// TIA Portal project "Proyecto_Automatizacion" (V18)

(* hardware
DEVICE "S7-1500/ET200MP station_1"  S7-1500 station
   slot 0: "Rail_0"  Rack  6ES7 590-1***0-0AA0
   slot 1: "Celda_Mecanizado"  CPU 1516-3 PN/DP  6ES7 516-3AN00-0AB0  V1.8
      slot 3: "CPU display_1"  6ES7591-1BA00-0AA0
      slot 32768: "PROFINET interface_1"  X1
         slot 32769: "Port_1"  X1 P1
         slot 32770: "Port_2"  X1 P2
      slot 33024: "PROFINET interface_2"  X2
         slot 33025: "Port_1"  X2 P1
      slot 33280: "DP interface_1"  X3
   slot 2: "DI 16x24VDC BA_1"  DI 16x24VDC BA  6ES7 521-1BH10-0AA0  V1.1
   slot 3: "DQ 8x24VDC/2A HF_1"  DQ 8x24VDC/2A HF  6ES7 522-1BF00-0AB0  V2.2
   slot 4: "AI 16xI BA_1"  AI 16xI BA  6ES7 531-7MH00-0AB0  V1.0
   slot 5: "AQ 2xU/I ST_1"  AQ 2xU/I ST  6ES7 532-5NB00-0AB0  V1.0
*)

// ===== PLC "Celda_Mecanizado"  CPU 1516-3 PN/DP =====

VAR_GLOBAL   // PLC tag table "Default tag table"
   "ON" AT %M0.0 : Bool;
   "OFF" AT %M0.1 : Bool;
   "SU" AT %M0.2 : Bool;
   "PP_ACINTA" AT %M0.3 : Bool;
   "NOTHING" AT %M0.4 : Bool;
   "V_RAW" AT %MW10 : Int;
   "REARME_LOCAL" AT %M0.5 : Bool;
   "REARME_GLOBAL" AT %M0.6 : Bool;
   "EMER" AT %M0.7 : Bool;
   "APAGADO" AT %M1.0 : Bool;
   "M_ACE" AT %M1.1 : Bool;
   "M_PAR" AT %M1.2 : Bool;
   "M_FR" AT %M1.3 : Bool;
   "CINTA_OFF" AT %M1.4 : Bool;
   "ERROR_L" AT %M1.5 : Bool;
   "ERROR_G" AT %M1.6 : Bool;
   "P_AS" AT %M1.7 : Bool;
   "P_S" AT %M2.0 : Bool;
   "AUTO" AT %M2.1 : Bool;
   "ERR_AUTO" AT %M2.2 : Bool;
   "CINTA_ON" AT %M2.3 : Bool;
   "CINTA_OK" AT %M2.4 : Bool;
   "CINTA_APAGAR" AT %M2.5 : Bool;
   "CINTA_CONG" AT %M2.6 : Bool;
   "MANT" AT %M2.7 : Bool;
END_VAR

DATA_BLOCK "Datos_Generales"   // DB1
{ S7_Optimized_Access := 'TRUE' }
VERSION : 0.1
   VAR
      Tiempo_Lim_Espada : Time := T#60s;
      Tiempo_Lim_Cuchillo : Time := T#60s;
      Tiempo_Lim_Katana : Time := T#60s;
      Tiempo_Lim_Florete : Time := T#60s;
      Tiempo_Lim_Sable : Time := T#60s;
      Tiempo_Lim_Hacha : Time := T#60s;
      Tiempo_Lim_Guada : Time := T#60s;
      Tiempo_Lim_MC : Time := T#60s;
      Tiempo_Lim_ML : Time := T#60s;
   END_VAR
BEGIN
END_DATA_BLOCK

FUNCTION_BLOCK "Interrupcion"   // FB1, STL
TITLE = Bloque de interrupción en la cinta
{ S7_Optimized_Access := 'TRUE' }
VERSION : 0.1
// Esta secuencia se ejecutará siempre que el robot Pick and Place quiera coger o dejar una pieza en la cinta.
   VAR_INPUT
      RESET : Bool;   // Evento asíncrono de prioridad máxima para la desconexión del bloque.
      C_PARADA : Bool;   // Indica que la cinta está completamente parada. Se recomienda que sea un sensor de velocidad que marque 0.
      FIN_INTERRUPCION : Bool;   // Indica que la interrupción ha finalizado y se vuelve al ciclo normal.
      TIEMPO_LIM : Time;   // Tiempo límite para la parada, si se sobrepasa dará error.
   END_VAR
   VAR_OUTPUT
      M_PARAR : Bool;   // Para la cinta de forma suave, con una rampa de frenado.
      B_FIN : Bool;   // Indica el fin de la interrupción y vuelta al ciclo normal.
      ERROR_PARADA : Bool;   // Indica que la cinta ha tardado mucho en parar. Ha habido un error.
      M_ACELERAR : Bool;   // Acelerar el motor.
      CINTA_PARADA : Bool;   // Acuse de recibo de cinta parada.
   END_VAR
   VAR
      B_TRABAJO : Bool;   // Bit de trabajo que controla la consexión por flanco
      X_PARADA : Bool;   // Etapa en la que se realiza la rampa de frenado.
      X_ESPERA : Bool;   // Etapa de espera hasta el fin de la interrupción.
      X_MOTOR : Bool;   // Etapa en la que se acelera el motor para evitar que se vuelva a tratar la misma pieza.
      AVISO_ERROR : Bool;   // Aviso interno del error de parada por tiempo excesivo.
      PARADA_REALIZADA : Bool;   // Se ha detenido el motor.
      MOTOR_OK : Bool;   // El motor ha movido la pieza lo suficiente.
      X_FIN : Bool;   // Etapa de fin de la interrupción.
      IEC_Timer_0_MOTOR : TON_TIME;
      Maniobra_PARADA : "Maniobra";
   END_VAR
BEGIN

REGION Network 1: DESCONEXIÓN POR RESET
   // Evento asíncrono de prioridad máxima. Resetea el bloque y sale de él.
         A     #RESET;

         R     #B_TRABAJO;
         R     #AVISO_ERROR;
         R     #X_ESPERA;
         R     #X_PARADA;
         R     #X_MOTOR;
         R     #X_FIN;

         R     #M_ACELERAR;
         R     #B_FIN;
         R     #ERROR_PARADA;

         JCN   _RESET;

         CALL  #Maniobra_PARADA
         ( RESET        := TRUE,
           FIN_MANIOBRA := ,
           TIEMPO_LIM   := ,
           ACTUADOR     := #M_PARAR,
           B_FIN        := ,
           ERROR_TIEMPO :=
         );


         CALL  RESET_TIMER
         ( "TIMER" := #IEC_Timer_0_MOTOR
         );

   _RESET:NOP   0;

         A     #RESET;
         BEC;
END_REGION

REGION Network 2: DESCONEXIÓN POR ERROR DE TIEMPO
   // Evento síncrono de error por temporización
         A     #AVISO_ERROR;

         R     #B_TRABAJO;

         S     #ERROR_PARADA;

         R     #M_ACELERAR;

         JCN   _TIEMPO;

         CALL  #Maniobra_PARADA
         ( RESET        := TRUE,
           FIN_MANIOBRA := ,
           TIEMPO_LIM   := ,
           ACTUADOR     := #M_PARAR,
           B_FIN        := ,
           ERROR_TIEMPO :=
         );


         CALL  RESET_TIMER
         ( "TIMER" := #IEC_Timer_0_MOTOR
         );

   _TIEMPO:NOP   0;

         A     #AVISO_ERROR;
         R     #AVISO_ERROR;
         BEC;
END_REGION

REGION Network 3: DESCONEXIÓN POR FIN DE LA INTERRUPCIÓN
   // Fin de la interrupción natural.
         A     #X_FIN;

         R     #B_TRABAJO;

         S     #B_FIN;

         R     #M_ACELERAR;

         JCN   _FIN;

         CALL  #Maniobra_PARADA
         ( RESET        := TRUE,
           FIN_MANIOBRA := ,
           TIEMPO_LIM   := ,
           ACTUADOR     := #M_PARAR,
           B_FIN        := ,
           ERROR_TIEMPO :=
         );


         CALL  RESET_TIMER
         ( "TIMER" := #IEC_Timer_0_MOTOR
         );

   _FIN: NOP   0;

         A     #X_FIN;
         R     #X_FIN;
         BEC;
END_REGION

REGION Network 4: CONEXIÓN DE LA INTERRUPCIÓN
         SET;
         FP    #B_TRABAJO;

         S     #X_PARADA;
         R     #X_FIN;
         R     #X_ESPERA;
         R     #X_MOTOR;
         R     #AVISO_ERROR;

         R     #ERROR_PARADA;
         R     #B_FIN;
END_REGION

REGION Network 5: CONTROL DEL TIEMPO DEL MOTOR
   // Se mide el tiempo necesario para que la pieza deje de estar delante del sensor y pueda volver al régimen permanente.
   // Se trata de un tiempo fijo no modificable, por lo que se pone directamente.
         CALL  #IEC_Timer_0_MOTOR
         ( IN := #X_MOTOR,
           PT := T#5s,
           Q  := #MOTOR_OK,
           ET :=
         );
END_REGION

REGION Network 6: PASO A ESPERA
   // Paso a la etapa de espera si la cinta se ha parado.
         A     #X_PARADA;

         JCN   _PARADA;
         CALL  #Maniobra_PARADA
         ( RESET        := FALSE,
           FIN_MANIOBRA := #C_PARADA,
           TIEMPO_LIM   := #TIEMPO_LIM,
           ACTUADOR     := #M_PARAR,
           B_FIN        := #PARADA_REALIZADA,
           ERROR_TIEMPO := #AVISO_ERROR
         );


         A     #PARADA_REALIZADA;

         S     #X_ESPERA;
         R     #X_PARADA;

   _PARADA:NOP   0;
END_REGION

REGION Network 7: PASO A MOVIMIENTO
   // Una vez a terminado la acción se mueve la cinta para evitar tratar de nuevo la misma pieza
         A     #X_ESPERA;
         A     #FIN_INTERRUPCION;

         S     #X_MOTOR;
         R     #X_ESPERA;
END_REGION

REGION Network 8: PASO A FIN
   // Paso a la etapa de fin si la interrupción se ha terminado.
         A     #X_MOTOR;
         A     #MOTOR_OK;

         S     #X_FIN;
         R     #X_MOTOR;
END_REGION

REGION Network 9: TRATAMIENTO DE ESPERA
   // Tratamiento de la etapa de espera.
         A     #X_ESPERA;
         =     #CINTA_PARADA;
END_REGION

REGION Network 10: TRATAMIENTO DEL MOVIMIENTO
   // Tratamiento de la etapa de movimiento.
         A     #X_MOTOR;
         =     #M_ACELERAR;
END_REGION
END_FUNCTION_BLOCK

FUNCTION_BLOCK "Cinta"   // FB2, STL
TITLE = BLOQUE DE LA CINTA
{ S7_Optimized_Access := 'TRUE' }
VERSION : 0.1
// Este bloque controlará las desconxeiones por petición y error, la conexión, el régimen permanente y las interrupciones de la cinta.
   VAR_INPUT
      PETICION_CONEXION : Bool;   // Petición de conexión de la Cinta.
      PETICION_DESCONEXION : Bool;   // Petición de desconexión de la cinta.
      VELOCIDAD_RAW : Int;   // Entrada de velocidad de la cinta analógica.
      V_med : Real;   // Velocidad deseada en régimen permanente.
      V_MIN : Real;   // Mínimo de velocidad que se puede medir.
      V_MAX : Real;   // Máximo de velocidad que se puede medir.
      V_MAX_ADM : Real;   // Máxima velocidad admitida en régimen permanente.
      V_MIN_ADM : Real;   // Mínima velocidad permitida en régimen permanente.
      SU : Bool;   // Sensor de presencia ultrasonido para detectar las cajas vacías
      PP_A_CINTA : Bool;   // Aviso de que el Pick and Place quiere dejar algo en la cinta.
      DO_NOTHING : Bool;   // Aviso de que la pieza detectada no requiere operación.
      TIEMPO_LIM : Time;   // Tiempo límite de regulación de velocidad.
      TIEMPO_LIM_ERROR_INT : Time;   // Tiempo límite para error de interrupción.
      REARME_LOCAL : Bool;   // Rearme local de la cinta.
      REARME : Bool;   // Rearme global tras emergencia asíncrona.
      EMER : Bool;   // Emergencia asíncrona.
      MANT : Bool;   // Petición de congelación de la cinta por mantenimiento.
      APAGADO_CONFIRMADO : Bool;   // Apagado de la cinta confirmado.
      ERROR_AUTO_DIAG : Bool;   // Error encontrado en el autodiagnóstico.
      CINTA_OK : Bool;   // Autodiagnóstico correcto.
   END_VAR
   VAR_OUTPUT
      M_ACELERAR : Bool;   // Señal de aceleración del motor.
      M_FRENAR : Bool;   // Señal de frenada del motor.
      M_PARAR : Bool;   // Señal de parada suave mediante rampa de frenado.
      PARADA_ASINCRONA : Bool;   // Señal de parada brusca por emergecia asíncrona.
      PARADA_SINCRONA : Bool;   // Señal de parada brusca por emergencia síncrona..
      CINTA_ON : Bool;   // Acuse de recibo de puesta en marcha.
      CINTA_OFF : Bool;   // Acuse de recibo de apagado.
      CINTA_CONG : Bool;   // Acuse de recibo de parada por mantenimiento.
      AUTO_DIAG_CINTA : Bool;   // Señal de autodiagnóstico de la cinta
      CINTA_APAGAR : Bool;   // Orden de apagado de la cinta.
      ERROR_GLOBAL : Bool;   // Chivato de error global.
      ERROR_LOCAL : Bool;   // Chivato de error local.
      CINTA_PARADA : Bool;   // Indica que la cinta está completamente parada para la carga y descarga.
   END_VAR
   VAR
      B_TRABAJO : Bool;   // Bit que indica si la cinta ya estaba encendida.
      X_ERROR_LOCAL : Bool;   // Etapa pozo por error local.
      X_EMER_GLOBAL : Bool;   // Etapa pozo por emergencia global.
      X1 : Bool;   // Etapa de autodiagnóstico.
      X2 : Bool;   // Etapa de aceleración inicial.
      X3 : Bool;   // Régimen permanente de velocidad.
      X4 : Bool;   // Etapa de frenado.
      X5 : Bool;   // Etapa de aceleración.
      XM1 : Bool;   // Macroetapa de interrupción por nueva pieza.
      XM2 : Bool;   // Macroetapa de interrupción por pieza terminadad.
      X10 : Bool;   // Etapa de solicitud a la desconexión natural.
      X_FIN : Bool;   // Apagado de la cinta.
      ERROR_PARADA : Bool;   // Error durante la parada de la cinta.
      C_FIN_INT1 : Bool;   // Conector para el fin de la interrupción 1.
      C_INI_INT2 : Bool;   // Conector para el inicio de la interrupción 2.
      ERROR_TEMPORIZACION : Bool;   // Error debido a exceso de tiempo.
      ERROR_MEDICION : Bool;   // Error durante la medición de la velocidad.
      Marcha_Motor_X2 : "Maniobra";
      Marcha_Motor_X4 : "Maniobra";
      Marcha_Motor_X5 : "Maniobra";
      Marcha_Motor_PARADA : "Maniobra";
      Interrupcion_PIEZA_NUEVA : "Interrupcion";
      Interrupcion_PIEZA_TERMINADA : "Interrupcion";
   END_VAR
   VAR_TEMP
      V_baja : Bool;   // La velocidad es muy lenta.
      V_alta : Bool;   // La velocidad es muy rápida.
      V_parada : Bool;   // Está parado.
      V_REAL : Real;   // Valor convertido de la velocidad.
      V_OK_SUBIDA : Bool;   // Velocidad alcanzada acelerando.
      V_OK_BAJADA : Bool;   // Velocidad alcanzada frenando.
      FIN_INT : Bool;   // Fin interrupción.
      FIN_MAN : Bool;   // Fin de la maniobra.
      FIN_PARADA : Bool;   // Fin de la parada.
   END_VAR
BEGIN

REGION Network 1: DESCONEXIÓN NORMAL
   // Desconexión de la cinta porque no se ha encendido todavía.
         AN    #PETICION_CONEXION;

         R     #B_TRABAJO;

         R     #CINTA_OFF;
         R     #CINTA_ON;
         R     #AUTO_DIAG_CINTA;

         JCN   _DESCONEXION;

         CALL  #Marcha_Motor_X2
         ( RESET        := TRUE,
           FIN_MANIOBRA := ,
           TIEMPO_LIM   := ,
           ACTUADOR     := #M_ACELERAR,
           B_FIN        := ,
           ERROR_TIEMPO :=
         );

         CALL  #Marcha_Motor_X4
         ( RESET        := TRUE,
           FIN_MANIOBRA := ,
           TIEMPO_LIM   := ,
           ACTUADOR     := #M_FRENAR,
           B_FIN        := ,
           ERROR_TIEMPO :=
         );

         CALL  #Marcha_Motor_X5
         ( RESET        := TRUE,
           FIN_MANIOBRA := ,
           TIEMPO_LIM   := ,
           ACTUADOR     := #M_ACELERAR,
           B_FIN        := ,
           ERROR_TIEMPO :=
         );

         CALL  #Marcha_Motor_PARADA
         ( RESET        := TRUE,
           FIN_MANIOBRA := ,
           TIEMPO_LIM   := ,
           ACTUADOR     := #CINTA_APAGAR,
           B_FIN        := ,
           ERROR_TIEMPO :=
         );

         CALL  #Interrupcion_PIEZA_NUEVA
         ( RESET            := TRUE,
           C_PARADA         := ,
           FIN_INTERRUPCION := ,
           TIEMPO_LIM       := ,
           M_PARAR          := #M_PARAR,
           B_FIN            := ,
           ERROR_PARADA     := ,
           M_ACELERAR       := #M_ACELERAR,
           CINTA_PARADA     := #CINTA_PARADA
         );

         CALL  #Interrupcion_PIEZA_TERMINADA
         ( RESET            := TRUE,
           C_PARADA         := ,
           FIN_INTERRUPCION := ,
           TIEMPO_LIM       := ,
           M_PARAR          := #M_PARAR,
           B_FIN            := ,
           ERROR_PARADA     := ,
           M_ACELERAR       := #M_ACELERAR,
           CINTA_PARADA     := #CINTA_PARADA
         );


   _DESCONEXION:NOP   0;
END_REGION

REGION Network 2: DESCONEXIÓN POR EMERGENCIA GLOBAL
   // Desconexión debida al error global.
         A     #X_EMER_GLOBAL;

         S     #PARADA_ASINCRONA;
         S     #ERROR_GLOBAL;
         R     #PARADA_SINCRONA;
         R     #CINTA_OFF;
         R     #CINTA_ON;
         R     #AUTO_DIAG_CINTA;

         JCN   _ERRGL;

         CALL  #Marcha_Motor_X2
         ( RESET        := TRUE,
           FIN_MANIOBRA := ,
           TIEMPO_LIM   := ,
           ACTUADOR     := #M_ACELERAR,
           B_FIN        := ,
           ERROR_TIEMPO :=
         );

         CALL  #Marcha_Motor_X4
         ( RESET        := TRUE,
           FIN_MANIOBRA := ,
           TIEMPO_LIM   := ,
           ACTUADOR     := #M_FRENAR,
           B_FIN        := ,
           ERROR_TIEMPO :=
         );

         CALL  #Marcha_Motor_X5
         ( RESET        := TRUE,
           FIN_MANIOBRA := ,
           TIEMPO_LIM   := ,
           ACTUADOR     := #M_ACELERAR,
           B_FIN        := ,
           ERROR_TIEMPO :=
         );

         CALL  #Marcha_Motor_PARADA
         ( RESET        := TRUE,
           FIN_MANIOBRA := ,
           TIEMPO_LIM   := ,
           ACTUADOR     := #CINTA_APAGAR,
           B_FIN        := ,
           ERROR_TIEMPO :=
         );

         CALL  #Interrupcion_PIEZA_NUEVA
         ( RESET            := TRUE,
           C_PARADA         := ,
           FIN_INTERRUPCION := ,
           TIEMPO_LIM       := ,
           M_PARAR          := #M_PARAR,
           B_FIN            := ,
           ERROR_PARADA     := ,
           M_ACELERAR       := #M_ACELERAR,
           CINTA_PARADA     := #CINTA_PARADA
         );

         CALL  #Interrupcion_PIEZA_TERMINADA
         ( RESET            := TRUE,
           C_PARADA         := ,
           FIN_INTERRUPCION := ,
           TIEMPO_LIM       := ,
           M_PARAR          := #M_PARAR,
           B_FIN            := ,
           ERROR_PARADA     := ,
           M_ACELERAR       := #M_ACELERAR,
           CINTA_PARADA     := #CINTA_PARADA
         );



   _ERRGL:NOP   0;
END_REGION

REGION Network 3: DESCONEXION ERROR LOCAL
   // Desconexión debida a un error local en la cinta, ya sea por el control de velocidad o durante el autodiagnóstico.
         A     #X_ERROR_LOCAL;

         R     #PARADA_ASINCRONA;
         S     #ERROR_LOCAL;
         S     #PARADA_SINCRONA;
         R     #CINTA_OFF;
         R     #CINTA_ON;
         R     #AUTO_DIAG_CINTA;

         JCN   _ERRLO;

         CALL  #Marcha_Motor_X2
         ( RESET        := TRUE,
           FIN_MANIOBRA := ,
           TIEMPO_LIM   := ,
           ACTUADOR     := #M_ACELERAR,
           B_FIN        := ,
           ERROR_TIEMPO :=
         );

         CALL  #Marcha_Motor_X4
         ( RESET        := TRUE,
           FIN_MANIOBRA := ,
           TIEMPO_LIM   := ,
           ACTUADOR     := #M_FRENAR,
           B_FIN        := ,
           ERROR_TIEMPO :=
         );

         CALL  #Marcha_Motor_X5
         ( RESET        := TRUE,
           FIN_MANIOBRA := ,
           TIEMPO_LIM   := ,
           ACTUADOR     := #M_ACELERAR,
           B_FIN        := ,
           ERROR_TIEMPO :=
         );

         CALL  #Marcha_Motor_PARADA
         ( RESET        := TRUE,
           FIN_MANIOBRA := ,
           TIEMPO_LIM   := ,
           ACTUADOR     := #CINTA_APAGAR,
           B_FIN        := ,
           ERROR_TIEMPO :=
         );

         CALL  #Interrupcion_PIEZA_NUEVA
         ( RESET            := TRUE,
           C_PARADA         := ,
           FIN_INTERRUPCION := ,
           TIEMPO_LIM       := ,
           M_PARAR          := #M_PARAR,
           B_FIN            := ,
           ERROR_PARADA     := ,
           M_ACELERAR       := #M_ACELERAR,
           CINTA_PARADA     := #CINTA_PARADA
         );

         CALL  #Interrupcion_PIEZA_TERMINADA
         ( RESET            := TRUE,
           C_PARADA         := ,
           FIN_INTERRUPCION := ,
           TIEMPO_LIM       := ,
           M_PARAR          := #M_PARAR,
           B_FIN            := ,
           ERROR_PARADA     := ,
           M_ACELERAR       := #M_ACELERAR,
           CINTA_PARADA     := #CINTA_PARADA
         );



   _ERRLO:NOP   0;
END_REGION

REGION Network 4: CONEXIÓN
         A     #PETICION_CONEXION;
         FP    #B_TRABAJO;

         S     #X1;
         R     #X2;
         R     #X3;
         R     #X4;
         R     #X5;
         R     #XM1;
         R     #XM2;
         R     #X10;
         R     #X_EMER_GLOBAL;
         R     #X_ERROR_LOCAL;
         R     #X_FIN;

         R     #ERROR_MEDICION;
         R     #ERROR_PARADA;
         R     #ERROR_TEMPORIZACION;

         R     #PARADA_ASINCRONA;
         R     #PARADA_SINCRONA;
         R     #ERROR_GLOBAL;
         R     #ERROR_LOCAL;
         R     #AUTO_DIAG_CINTA;
         R     #CINTA_OFF;
         R     #CINTA_ON;

         JCN   _CONEXION;

         CALL  #Marcha_Motor_X2
         ( RESET        := TRUE,
           FIN_MANIOBRA := ,
           TIEMPO_LIM   := ,
           ACTUADOR     := #M_ACELERAR,
           B_FIN        := ,
           ERROR_TIEMPO :=
         );

         CALL  #Marcha_Motor_X4
         ( RESET        := TRUE,
           FIN_MANIOBRA := ,
           TIEMPO_LIM   := ,
           ACTUADOR     := #M_FRENAR,
           B_FIN        := ,
           ERROR_TIEMPO :=
         );

         CALL  #Marcha_Motor_X5
         ( RESET        := TRUE,
           FIN_MANIOBRA := ,
           TIEMPO_LIM   := ,
           ACTUADOR     := #M_ACELERAR,
           B_FIN        := ,
           ERROR_TIEMPO :=
         );

         CALL  #Marcha_Motor_PARADA
         ( RESET        := TRUE,
           FIN_MANIOBRA := ,
           TIEMPO_LIM   := ,
           ACTUADOR     := #CINTA_APAGAR,
           B_FIN        := ,
           ERROR_TIEMPO :=
         );

         CALL  #Interrupcion_PIEZA_NUEVA
         ( RESET            := TRUE,
           C_PARADA         := ,
           FIN_INTERRUPCION := ,
           TIEMPO_LIM       := ,
           M_PARAR          := #M_PARAR,
           B_FIN            := ,
           ERROR_PARADA     := ,
           M_ACELERAR       := #M_ACELERAR,
           CINTA_PARADA     := #CINTA_PARADA
         );

         CALL  #Interrupcion_PIEZA_TERMINADA
         ( RESET            := TRUE,
           C_PARADA         := ,
           FIN_INTERRUPCION := ,
           TIEMPO_LIM       := ,
           M_PARAR          := #M_PARAR,
           B_FIN            := ,
           ERROR_PARADA     := ,
           M_ACELERAR       := #M_ACELERAR,
           CINTA_PARADA     := #CINTA_PARADA
         );



   _CONEXION:NOP   0;
END_REGION

REGION Network 5: CONGELACIÓN
   // Congelación de la cinta por matenimiento.
         A     #MANT;

         =     #CINTA_CONG;
         R     #AUTO_DIAG_CINTA;

         JCN   _CONGELACION;

         CALL  #Marcha_Motor_X2
         ( RESET        := TRUE,
           FIN_MANIOBRA := ,
           TIEMPO_LIM   := ,
           ACTUADOR     := #M_ACELERAR,
           B_FIN        := ,
           ERROR_TIEMPO :=
         );

         CALL  #Marcha_Motor_X4
         ( RESET        := TRUE,
           FIN_MANIOBRA := ,
           TIEMPO_LIM   := ,
           ACTUADOR     := #M_FRENAR,
           B_FIN        := ,
           ERROR_TIEMPO :=
         );

         CALL  #Marcha_Motor_X5
         ( RESET        := TRUE,
           FIN_MANIOBRA := ,
           TIEMPO_LIM   := ,
           ACTUADOR     := #M_ACELERAR,
           B_FIN        := ,
           ERROR_TIEMPO :=
         );

         CALL  #Marcha_Motor_PARADA
         ( RESET        := TRUE,
           FIN_MANIOBRA := ,
           TIEMPO_LIM   := ,
           ACTUADOR     := #CINTA_APAGAR,
           B_FIN        := ,
           ERROR_TIEMPO :=
         );

         CALL  #Interrupcion_PIEZA_NUEVA
         ( RESET            := TRUE,
           C_PARADA         := ,
           FIN_INTERRUPCION := ,
           TIEMPO_LIM       := ,
           M_PARAR          := #M_PARAR,
           B_FIN            := ,
           ERROR_PARADA     := ,
           M_ACELERAR       := #M_ACELERAR,
           CINTA_PARADA     := #CINTA_PARADA
         );

         CALL  #Interrupcion_PIEZA_TERMINADA
         ( RESET            := TRUE,
           C_PARADA         := ,
           FIN_INTERRUPCION := ,
           TIEMPO_LIM       := ,
           M_PARAR          := #M_PARAR,
           B_FIN            := ,
           ERROR_PARADA     := ,
           M_ACELERAR       := #M_ACELERAR,
           CINTA_PARADA     := #CINTA_PARADA
         );


   _CONGELACION:NOP   0;

         A     #MANT;
         BEC;
END_REGION

REGION Network 6: REARME GLOBAL
   // Rearme tras emergencia global.
         A     #X_EMER_GLOBAL;
         A     #REARME;

         R     #X_EMER_GLOBAL;
         R     #B_TRABAJO;
END_REGION

REGION Network 7: REARME LOCAL
   // Rearme tras emergencia local.
         A     #X_ERROR_LOCAL;
         A     #REARME_LOCAL;

         R     #X_ERROR_LOCAL;
         R     #B_TRABAJO;
END_REGION

REGION Network 8: CONECTORES
   // Tratamiento de todos los conectores necesarios (velocidad y tiempos límite).
         CALL  "Tratamiento_velocidad"
         ( V_RAW       := #VELOCIDAD_RAW,
           V_med       := #V_med,
           V_MIN       := #V_MIN,
           V_MAX       := #V_MAX,
           V_MAX_ADM   := #V_MAX_ADM,
           V_MIN_ADM   := #V_MIN_ADM,
           V_baja      := #V_baja,
           V_alta      := #V_alta,
           V_parada    := #V_parada,
           V_OK_SUBIDA := #V_OK_SUBIDA,
           V_OK_BAJADA := #V_OK_BAJADA,
           V_REAL      := #V_REAL,
           ERROR       := #ERROR_MEDICION
         );

   // Conector de fin de interrupción 1
         AN    #SU;
         O     #DO_NOTHING;
         =     #C_FIN_INT1;

   // Conector de inicio de interrupción 2
         AN    #SU;
         A     #PP_A_CINTA;
         =     #C_INI_INT2;
END_REGION

REGION Network 9: ERROR GLOBAL
   // Salto a etapa de emergencia global.
         A     #EMER;

         S     #X_EMER_GLOBAL;
         R     #X1;
         R     #X2;
         R     #X3;
         R     #X4;
         R     #X5;
         R     #XM1;
         R     #XM2;
END_REGION

REGION Network 10: ERROR LOCAL
   // Salto a etapa de emergencia local.
         A     #ERROR_AUTO_DIAG;
         O     #ERROR_MEDICION;
         O     #ERROR_PARADA;
         O     #ERROR_TEMPORIZACION;
         O(;
         A     #X3;
         A     #V_parada;
         );

         S     #X_ERROR_LOCAL;
         R     #XM1;
         R     #XM2;
         R     #X1;
         R     #X2;
         R     #X3;
         R     #X4;
         R     #X5;
END_REGION

REGION Network 11: CINTA ENCENDIDA (X1 -> X2)
   // La cinta se pone en marcha tras el autodiagnóstico.
         A     #X1;
         A     #CINTA_OK;

         S     #X2;
         R     #X1;
END_REGION

REGION Network 12: X2 -> X3
   // La cinta llega al régimen permanente
         A     #X2;

         JCN   _X2;

         CALL  #Marcha_Motor_X2
         ( RESET        := FALSE,
           FIN_MANIOBRA := #V_OK_SUBIDA,
           TIEMPO_LIM   := #TIEMPO_LIM,
           ACTUADOR     := #M_ACELERAR,
           B_FIN        := #FIN_MAN,
           ERROR_TIEMPO := #ERROR_TEMPORIZACION
         );

         A     #FIN_MAN;
         S     #X3;
         R     #X2;

   _X2:  NOP   0;
END_REGION

REGION Network 13: X3 -> X4
   // La cinta pierde velocidad.
         A     #X3;
         A     #V_alta;

         S     #X4;
         R     #X3;
END_REGION

REGION Network 14: X3 -> X5
   // La cinta gana velocidad.
         A     #X3;
         A     #V_baja;

         S     #X5;
         R     #X3;
END_REGION

REGION Network 15: X4 -> X3
   // Vuelta al régimen permanente.
         A     #X4;
         JCN   _X4;

         CALL  #Marcha_Motor_X4
         ( RESET        := FALSE,
           FIN_MANIOBRA := #V_OK_BAJADA,
           TIEMPO_LIM   := #TIEMPO_LIM,
           ACTUADOR     := #M_FRENAR,
           B_FIN        := #FIN_MAN,
           ERROR_TIEMPO := #ERROR_TEMPORIZACION
         );

         A     #FIN_MAN;
         S     #X3;
         R     #X4;

   _X4:  NOP   0;
END_REGION

REGION Network 16: X5 ->X3
   // Vuelta al régimen permanente.
         A     #X5;
         JCN   _X5;

         CALL  #Marcha_Motor_X5
         ( RESET        := FALSE,
           FIN_MANIOBRA := #V_OK_SUBIDA,
           TIEMPO_LIM   := #TIEMPO_LIM,
           ACTUADOR     := #M_ACELERAR,
           B_FIN        := #FIN_MAN,
           ERROR_TIEMPO := #ERROR_TEMPORIZACION
         );

         A     #FIN_MAN;
         S     #X3;
         R     #X5;

   _X5:  NOP   0;
END_REGION

REGION Network 17: INTERRUPCION 1 (XM1)
         A(;
         O     #X2;
         O     #X3;
         O     #X4;
         O     #X5;
         );
         A     #SU;

         S     #XM1;
         R     #X2;
         R     #X3;
         R     #X4;
         R     #X5;
END_REGION

REGION Network 18: TRATAMIENTO DE INTERRUPCION 1 (XM1)
         A     #XM1;

         JCN   _INTERRUPCION_1;

   // Interrumpir los procesos que se estén ejecutando
         CALL  #Marcha_Motor_X2
         ( RESET        := TRUE,
           FIN_MANIOBRA := ,
           TIEMPO_LIM   := ,
           ACTUADOR     := #M_ACELERAR,
           B_FIN        := ,
           ERROR_TIEMPO :=
         );

         CALL  #Marcha_Motor_X4
         ( RESET        := TRUE,
           FIN_MANIOBRA := ,
           TIEMPO_LIM   := ,
           ACTUADOR     := #M_FRENAR,
           B_FIN        := ,
           ERROR_TIEMPO :=
         );

         CALL  #Marcha_Motor_X5
         ( RESET        := TRUE,
           FIN_MANIOBRA := ,
           TIEMPO_LIM   := ,
           ACTUADOR     := #M_ACELERAR,
           B_FIN        := ,
           ERROR_TIEMPO :=
         );

   // Ejecutar la interrupción
         CALL  #Interrupcion_PIEZA_NUEVA
         ( RESET            := FALSE,
           C_PARADA         := #V_parada,
           FIN_INTERRUPCION := #C_FIN_INT1,
           TIEMPO_LIM       := #TIEMPO_LIM_ERROR_INT,
           M_PARAR          := #M_PARAR,
           B_FIN            := #FIN_INT,
           ERROR_PARADA     := #ERROR_PARADA,
           M_ACELERAR       := #M_ACELERAR,
           CINTA_PARADA     := #CINTA_PARADA
         );

         A     #FIN_INT;

         S     #X2;
         R     #XM1;

         A     #ERROR_PARADA;

         S     #X_ERROR_LOCAL;
         R     #XM1;

   _INTERRUPCION_1:NOP   0;
END_REGION

REGION Network 19: INTERRUPCION 2 (XM2)
         A(;
         O     #X2;
         O     #X3;
         O     #X4;
         O     #X5;
         );
         A     #C_INI_INT2;

         S     #XM2;
         R     #X2;
         R     #X3;
         R     #X4;
         R     #X5;
END_REGION

REGION Network 20: TRATAMIENTO DE INTERRUPCION 2 (XM2)
         A     #XM2;

         JCN   _INTERRUPCION_2;

   // Interrumpir los procesos que se estén ejecutando
         CALL  #Marcha_Motor_X2
         ( RESET        := TRUE,
           FIN_MANIOBRA := ,
           TIEMPO_LIM   := ,
           ACTUADOR     := #M_ACELERAR,
           B_FIN        := ,
           ERROR_TIEMPO :=
         );

         CALL  #Marcha_Motor_X4
         ( RESET        := TRUE,
           FIN_MANIOBRA := ,
           TIEMPO_LIM   := ,
           ACTUADOR     := #M_FRENAR,
           B_FIN        := ,
           ERROR_TIEMPO :=
         );

         CALL  #Marcha_Motor_X5
         ( RESET        := TRUE,
           FIN_MANIOBRA := ,
           TIEMPO_LIM   := ,
           ACTUADOR     := #M_ACELERAR,
           B_FIN        := ,
           ERROR_TIEMPO :=
         );

   // Ejecutar la interrupción
         CALL  #Interrupcion_PIEZA_TERMINADA
         ( RESET            := FALSE,
           C_PARADA         := #V_parada,
           FIN_INTERRUPCION := #SU,
           TIEMPO_LIM       := #TIEMPO_LIM_ERROR_INT,
           M_PARAR          := #M_PARAR,
           B_FIN            := #FIN_INT,
           ERROR_PARADA     := #ERROR_PARADA,
           M_ACELERAR       := #M_ACELERAR,
           CINTA_PARADA     := #CINTA_PARADA
         );

         A     #FIN_INT;

         S     #X2;
         R     #XM2;

         A     #ERROR_PARADA;

         S     #X_ERROR_LOCAL;
         R     #XM2;

   _INTERRUPCION_2:NOP   0;
END_REGION

REGION Network 21: PETICION DE PARADA
         A     #PETICION_DESCONEXION;
         A(;
         O     #X1;
         O     #X2;
         O     #X3;
         O     #X4;
         O     #X5;
         );

         S     #X10;
         R     #X1;
         R     #X2;
         R     #X3;
         R     #X4;
         R     #X5;
END_REGION

REGION Network 22: TRATAMIENTO X1
         A     #X1;
         =     #AUTO_DIAG_CINTA;
         S     #CINTA_ON;
END_REGION

REGION Network 23: APAGADO DE LA CINTA.
         A     #X10;
         S     #CINTA_OFF;
         R     #CINTA_ON;
         JCN   _PARADA;

         CALL  #Marcha_Motor_X2
         ( RESET        := TRUE,
           FIN_MANIOBRA := ,
           TIEMPO_LIM   := ,
           ACTUADOR     := #M_ACELERAR,
           B_FIN        := ,
           ERROR_TIEMPO :=
         );

         CALL  #Marcha_Motor_X4
         ( RESET        := TRUE,
           FIN_MANIOBRA := ,
           TIEMPO_LIM   := ,
           ACTUADOR     := #M_FRENAR,
           B_FIN        := ,
           ERROR_TIEMPO :=
         );

         CALL  #Marcha_Motor_X5
         ( RESET        := TRUE,
           FIN_MANIOBRA := ,
           TIEMPO_LIM   := ,
           ACTUADOR     := #M_ACELERAR,
           B_FIN        := ,
           ERROR_TIEMPO :=
         );

         CALL  #Marcha_Motor_PARADA
         ( RESET        := FALSE,
           FIN_MANIOBRA := #APAGADO_CONFIRMADO,
           TIEMPO_LIM   := #TIEMPO_LIM,
           ACTUADOR     := #CINTA_APAGAR,
           B_FIN        := #FIN_PARADA,
           ERROR_TIEMPO := #ERROR_TEMPORIZACION
         );

         A     #FIN_PARADA;
         S     #X_FIN;
         R     #X10;

         A     #ERROR_TEMPORIZACION;
         S     #X_ERROR_LOCAL;
         R     #X10;

   _PARADA:NOP   0;
END_REGION
END_FUNCTION_BLOCK

FUNCTION_BLOCK "Maniobra"   // FB3, STL
TITLE = Bloque de velocidad en la cinta
{ S7_Optimized_Access := 'TRUE' }
VERSION : 0.1
// Esta secuencia se ejecutará siempre que la cinta deba moderar la velocidad.
   VAR_INPUT
      RESET : Bool;   // Evento asíncrono de prioridad máxima para la desconexión del bloque.
      FIN_MANIOBRA : Bool;   // Indica que la maniobra ha finalizado y se vuelve al ciclo normal.
      TIEMPO_LIM : Time;   // Tiempo límite para la maniobra, si se sobrepasa dará error.
   END_VAR
   VAR_OUTPUT
      ACTUADOR : Bool;   // Actúa sobre el actuador.
      B_FIN : Bool;   // Indica el fin de la maniobra y vuelta al ciclo normal.
      ERROR_TIEMPO : Bool;   // Indica que la cinta ha tardado mucho en parar. Ha habido un cambiar su velocidad.
   END_VAR
   VAR
      B_TRABAJO : Bool;   // Bit de trabajo que controla la consexión por flanco
      X_MARCHA : Bool;   // Etapa en la que se realiza la acción.
      AVISO_ERROR : Bool;   // Aviso interno del error de parada por tiempo excesivo.
      TEMP_ALTO : Bool;   // Salto del temporizador.
      X_FIN : Bool;   // Etapa de fin de la interrupción.
      IEC_Timer_Marcha : TON_TIME;
   END_VAR
BEGIN

REGION Network 1: DESCONEXIÓN POR RESET
   // Evento asíncrono de prioridad máxima. Resetea el bloque y sale de él.
         A     #RESET;

         R     #B_TRABAJO;
         R     #AVISO_ERROR;
         R     #X_MARCHA;
         R     #X_FIN;

         R     #ACTUADOR;
         R     #B_FIN;
         R     #ERROR_TIEMPO;

         JCN   _RESET;
         CALL  RESET_TIMER
         ( "TIMER" := #IEC_Timer_Marcha
         );
   _RESET:NOP   0;

         A     #RESET;
         BEC;
END_REGION

REGION Network 2: DESCONEXIÓN POR ERROR DE TIEMPO
   // Evento síncrono de error por temporización
         A     #AVISO_ERROR;

         R     #B_TRABAJO;

         S     #ERROR_TIEMPO;

         R     #ACTUADOR;

         JCN   _TIEMPO;
         CALL  RESET_TIMER
         ( "TIMER" := #IEC_Timer_Marcha
         );
   _TIEMPO:NOP   0;

         A     #AVISO_ERROR;
         R     #AVISO_ERROR;
         BEC;
END_REGION

REGION Network 3: DESCONEXIÓN POR FIN DE LA MARCHA
   // Fin de la marcha natural.
         A     #X_FIN;

         R     #B_TRABAJO;

         S     #B_FIN;

         R     #ACTUADOR;

         JCN   _FIN;
         CALL  RESET_TIMER
         ( "TIMER" := #IEC_Timer_Marcha
         );
   _FIN: NOP   0;

         A     #X_FIN;
         R     #X_FIN;
         BEC;
END_REGION

REGION Network 4: CONEXIÓN DE LA MARCHA
         SET;
         FP    #B_TRABAJO;

         S     #X_MARCHA;
         R     #X_FIN;
         R     #AVISO_ERROR;

         R     #ERROR_TIEMPO;
         R     #B_FIN;
END_REGION

REGION Network 5: ACTIVACIÓN DEL ERROR POR TIEMPO
   // Si se está demasiado tiempo en la etapa de parada se activa el aviso de error y se ejecuta la desconexión.
         CALL  #IEC_Timer_Marcha
         ( IN := #X_MARCHA,
           PT := #TIEMPO_LIM,
           Q  := #TEMP_ALTO,
           ET :=
         );


         A     #TEMP_ALTO;
         S     #AVISO_ERROR;
END_REGION

REGION Network 6: PASO A FIN
   // Paso a la etapa de fin si la interrupción se ha terminado.
         A     #X_MARCHA;
         A     #FIN_MANIOBRA;

         S     #X_FIN;
         R     #X_MARCHA;
END_REGION

REGION Network 7: TRATAMIENTO DE LA MARCHA
   // Tratamiento de la etapa de parada.
         A     #X_MARCHA;
         =     #ACTUADOR;
END_REGION
END_FUNCTION_BLOCK

FUNCTION_BLOCK "CNC"   // FB4, LAD
TITLE = BLOQUE CNC
{ S7_Optimized_Access := 'TRUE' }
VERSION : 0.1
// Este bloque se ejecutará para el control de la CNC.
   VAR_INPUT
      PETICION_CONEXION : Bool;   // Petición de conexión de la CNC.
      PETICION_APAGADO : Bool;   // Petición de desconexión de la CNC.
      LIQUIDO_RAW : Int;   // Entrada de nivel de refirgerante de la CNC analógica.
      L_crit : Real;   // Nivel crítico del líquido de refrigerante.
      L_MIN : Real;   // Mínimo de refrigerante que se puede medir.
      L_MAX : Real;   // Máximo de refirgerante que se puede medir.
      PIEZA_IN : Bool;   // Pieza dentro de la CNC.
      S_ESPADA : Bool;   // Detección de la espada.
      S_CUCHILLO : Bool;   // Detección del cuchillo.
      S_KATANA : Bool;   // Detección de la katana.
      S_FLORETE : Bool;   // Detección del florete.
      S_SABLE : Bool;   // Detección del sable.
      S_HACHA : Bool;   // Detección del hacha.
      S_GUADA : Bool;   // Detección de la guadaña.
      S_MC : Bool;   // Detección de mango corto.
      S_ML : Bool;   // Detección de mango largo.
      FIN_MEC : Bool;   // Fin del mecanizado.
      MANT : Bool;   // Petición de congelación por mantenimiento.
      EMER : Bool;   // Emergencia global asíncrona.
      REARME_LOCAL : Bool;   // Rearme local tras parada síncrona.
      REARME_GLOBAL : Bool;   // Rearme global tras parada asíncrona.
      APAGADO_CONFIRMADO : Bool;   // Confirmación del apagado de la CNC.
      ERROR_CNC : Bool;   // Error encontrado durante el autodiagnóstico de la CNC.
      OK_CNC : Bool;   // CNC ok tras autodiagnóstico.
      TIEMPO_LIM : Time;   // Tiempo límite para el apagado.
   END_VAR
   VAR_OUTPUT
      AUTO_DIAG_CNC : Bool;   // Señal de autodiagnóstico de la CNC.
      MEC_ESP : Bool;   // Mecanizado de la espada.
      MEC_CUC : Bool;   // Mecanizado del cuchillo.
      MEC_KAT : Bool;   // Mecanizado de la katana.
      MEC_FLO : Bool;   // Mecanizado del florete.
      MEC_SAB : Bool;   // Mecanizado del sable.
      MEC_HAC : Bool;   // Mecanizado del hacha.
      MEC_GUA : Bool;   // Mecanizado de la guadaña.
      MEC_MC : Bool;   // Mecanizado de mango corto.
      MEC_ML : Bool;   // Mecanizado de mango largo.
      APAGADO_CNC : Bool;   // Orden de apagado de la CNC.
      PARADA_SINCRONA : Bool;   // Señal de parada brusca por emergecia síncrona.
      PARADA_ASINCRONA : Bool;   // Señal de parada brusca por emergencia asíncrona.
      ERROR_REFRI : Bool;   // Chivato de error por refrigerante crítico.
      ERROR_TIEMPO : Bool;   // Chivato de error por límite de tiempo.
      ERROR_GLOBAL : Bool;   // Chivato de error global.
      ERROR_LOCAL : Bool;   // Chivato de error local por autodiagnóstico.
      ON_M : Bool;   // CNC conectada.
      OFF_M : Bool;   // CNC apagada.
      STANDBY_CNC : Bool;   // CNC en stan-by.
      CONG_M : Bool;   // Chivato de congelación de la CNC.
   END_VAR
   VAR
      B_TRABAJO : Bool;   // Bit que indica si la CNC ya estaba encendida.
      X21 : Bool;   // Etapa de autodiagnóstico.
      X22 : Bool;   // Etapa de espera (stand by).
      X23 : Bool;   // Etapa mecanizado de espada.
      X24 : Bool;   // Etapa mecanizado de cuchillo.
      X25 : Bool;   // Etapa mecanizado de katana.
      X26 : Bool;   // Etapa mecanizado de florete.
      X27 : Bool;   // Etapa mecanizado de sable.
      X28 : Bool;   // Etapa mecanizado de hacha.
      X29 : Bool;   // Etapa mecanizado de guadaña.
      X30 : Bool;   // Etapa mecanizado de mango corto.
      X31 : Bool;   // Etapa mecanizado de mango largo.
      X_APAGADO : Bool;   // Etapa de petición de apagado.
      X35 : Bool;   // Etapa de error global.
      X36 : Bool;   // Etapa de error por autodiagnóstico.
      X37 : Bool;   // Etapa de error por tiempo.
      X38 : Bool;   // Etapa de error por refrigerante.
      ERROR_MEDICION : Bool;   // Error durante la medición analógica.
      FLAG_REFRI : Bool;   // Flag del error del refirgerante.
      X_FIN : Bool;   // Apagado completo confirmado de la CNC.
      Maniobra_Espada : "Maniobra";
      Maniobra_cuchillo : "Maniobra";
      Maniobra_katana : "Maniobra";
      Maniobra_florete : "Maniobra";
      Maniobra_sable : "Maniobra";
      Maniobra_hacha : "Maniobra";
      Maniobra_ML : "Maniobra";
      Maniobra_IMC : "Maniobra";
      Maniobra_MC : "Maniobra";
      Maniobra_guada : "Maniobra";
      Maniobra_APAGADO : "Maniobra";
   END_VAR
   VAR_TEMP
      L_LIM : Bool;   // Limite de refrigerante alcanzado.
      L_REAL : Real;   // Valor convertido del refrigerante.
      FIN_MAN : Bool;   // Fin de la maniobra.
      FIN_PARADA : Bool;   // Fin de la parada.
   END_VAR
   VAR_TEMP   // added for the SCL form of the ladder/FBD networks
      _w1 : Bool;
   END_VAR
BEGIN

REGION Network 1 (STL): DESCONEXIÓN
   // Desconexión de la CNC si no es llamada.
         AN    #PETICION_CONEXION;

         R     #B_TRABAJO;

         R     #ON_M;
         R     #OFF_M;
         R     #AUTO_DIAG_CNC;

         JCN   _DESCONEXION;

         CALL  #Maniobra_Espada
         ( RESET        := TRUE,
           FIN_MANIOBRA := ,
           TIEMPO_LIM   := ,
           ACTUADOR     := #MEC_ESP,
           B_FIN        := ,
           ERROR_TIEMPO :=
         );

         CALL  #Maniobra_cuchillo
         ( RESET        := TRUE,
           FIN_MANIOBRA := ,
           TIEMPO_LIM   := ,
           ACTUADOR     := #MEC_CUC,
           B_FIN        := ,
           ERROR_TIEMPO :=
         );

         CALL  #Maniobra_katana
         ( RESET        := TRUE,
           FIN_MANIOBRA := ,
           TIEMPO_LIM   := ,
           ACTUADOR     := #MEC_KAT,
           B_FIN        := ,
           ERROR_TIEMPO :=
         );

         CALL  #Maniobra_florete
         ( RESET        := TRUE,
           FIN_MANIOBRA := ,
           TIEMPO_LIM   := ,
           ACTUADOR     := #MEC_FLO,
           B_FIN        := ,
           ERROR_TIEMPO :=
         );

         CALL  #Maniobra_sable
         ( RESET        := TRUE,
           FIN_MANIOBRA := ,
           TIEMPO_LIM   := ,
           ACTUADOR     := ,
           B_FIN        := #MEC_SAB,
           ERROR_TIEMPO :=
         );

         CALL  #Maniobra_hacha
         ( RESET        := TRUE,
           FIN_MANIOBRA := ,
           TIEMPO_LIM   := ,
           ACTUADOR     := ,
           B_FIN        := #MEC_HAC,
           ERROR_TIEMPO :=
         );

         CALL  #Maniobra_guada
         ( RESET        := TRUE,
           FIN_MANIOBRA := ,
           TIEMPO_LIM   := ,
           ACTUADOR     := ,
           B_FIN        := #MEC_GUA,
           ERROR_TIEMPO :=
         );

         CALL  #Maniobra_MC
         ( RESET        := TRUE,
           FIN_MANIOBRA := ,
           TIEMPO_LIM   := ,
           ACTUADOR     := ,
           B_FIN        := #MEC_MC,
           ERROR_TIEMPO :=
         );

         CALL  #Maniobra_ML
         ( RESET        := TRUE,
           FIN_MANIOBRA := ,
           TIEMPO_LIM   := ,
           ACTUADOR     := ,
           B_FIN        := #MEC_ML,
           ERROR_TIEMPO :=
         );


   _DESCONEXION:NOP   0;

         AN    #PETICION_CONEXION;
         BEC;
END_REGION

REGION Network 2 (STL): DESCONEXIÓN POR EMERGENCIA GLOBAL
   // Desconexión debida al error global.
         A     #X35;

         S     #PARADA_ASINCRONA;
         S     #ERROR_GLOBAL;
         R     #PARADA_SINCRONA;
         R     #OFF_M;
         R     #ON_M;
         R     #AUTO_DIAG_CNC;

         JCN   _ERRGL;
         CALL  #Maniobra_Espada
         ( RESET        := TRUE,
           FIN_MANIOBRA := ,
           TIEMPO_LIM   := ,
           ACTUADOR     := #MEC_ESP,
           B_FIN        := ,
           ERROR_TIEMPO :=
         );

         CALL  #Maniobra_cuchillo
         ( RESET        := TRUE,
           FIN_MANIOBRA := ,
           TIEMPO_LIM   := ,
           ACTUADOR     := #MEC_CUC,
           B_FIN        := ,
           ERROR_TIEMPO :=
         );

         CALL  #Maniobra_katana
         ( RESET        := TRUE,
           FIN_MANIOBRA := ,
           TIEMPO_LIM   := ,
           ACTUADOR     := #MEC_KAT,
           B_FIN        := ,
           ERROR_TIEMPO :=
         );

         CALL  #Maniobra_florete
         ( RESET        := TRUE,
           FIN_MANIOBRA := ,
           TIEMPO_LIM   := ,
           ACTUADOR     := #MEC_FLO,
           B_FIN        := ,
           ERROR_TIEMPO :=
         );

         CALL  #Maniobra_sable
         ( RESET        := TRUE,
           FIN_MANIOBRA := ,
           TIEMPO_LIM   := ,
           ACTUADOR     := ,
           B_FIN        := #MEC_SAB,
           ERROR_TIEMPO :=
         );

         CALL  #Maniobra_hacha
         ( RESET        := TRUE,
           FIN_MANIOBRA := ,
           TIEMPO_LIM   := ,
           ACTUADOR     := ,
           B_FIN        := #MEC_HAC,
           ERROR_TIEMPO :=
         );

         CALL  #Maniobra_guada
         ( RESET        := TRUE,
           FIN_MANIOBRA := ,
           TIEMPO_LIM   := ,
           ACTUADOR     := ,
           B_FIN        := #MEC_GUA,
           ERROR_TIEMPO :=
         );

         CALL  #Maniobra_MC
         ( RESET        := TRUE,
           FIN_MANIOBRA := ,
           TIEMPO_LIM   := ,
           ACTUADOR     := ,
           B_FIN        := #MEC_MC,
           ERROR_TIEMPO :=
         );

         CALL  #Maniobra_ML
         ( RESET        := TRUE,
           FIN_MANIOBRA := ,
           TIEMPO_LIM   := ,
           ACTUADOR     := ,
           B_FIN        := #MEC_ML,
           ERROR_TIEMPO :=
         );


   _ERRGL:NOP   0;
END_REGION

REGION Network 3 (STL): DESCONEXIÓN POR ERROR LOCAL EN CNC
   // Desconexión por error local en el autodiagnóstico.
         A     #X36;

         R     #PARADA_ASINCRONA;
         S     #ERROR_LOCAL;
         S     #PARADA_SINCRONA;
         R     #OFF_M;
         R     #ON_M;
         R     #AUTO_DIAG_CNC;

         JCN   _ERRLO;

         CALL  #Maniobra_Espada
         ( RESET        := TRUE,
           FIN_MANIOBRA := ,
           TIEMPO_LIM   := ,
           ACTUADOR     := #MEC_ESP,
           B_FIN        := ,
           ERROR_TIEMPO :=
         );

         CALL  #Maniobra_cuchillo
         ( RESET        := TRUE,
           FIN_MANIOBRA := ,
           TIEMPO_LIM   := ,
           ACTUADOR     := #MEC_CUC,
           B_FIN        := ,
           ERROR_TIEMPO :=
         );

         CALL  #Maniobra_katana
         ( RESET        := TRUE,
           FIN_MANIOBRA := ,
           TIEMPO_LIM   := ,
           ACTUADOR     := #MEC_KAT,
           B_FIN        := ,
           ERROR_TIEMPO :=
         );

         CALL  #Maniobra_florete
         ( RESET        := TRUE,
           FIN_MANIOBRA := ,
           TIEMPO_LIM   := ,
           ACTUADOR     := #MEC_FLO,
           B_FIN        := ,
           ERROR_TIEMPO :=
         );

         CALL  #Maniobra_sable
         ( RESET        := TRUE,
           FIN_MANIOBRA := ,
           TIEMPO_LIM   := ,
           ACTUADOR     := ,
           B_FIN        := #MEC_SAB,
           ERROR_TIEMPO :=
         );

         CALL  #Maniobra_hacha
         ( RESET        := TRUE,
           FIN_MANIOBRA := ,
           TIEMPO_LIM   := ,
           ACTUADOR     := ,
           B_FIN        := #MEC_HAC,
           ERROR_TIEMPO :=
         );

         CALL  #Maniobra_guada
         ( RESET        := TRUE,
           FIN_MANIOBRA := ,
           TIEMPO_LIM   := ,
           ACTUADOR     := ,
           B_FIN        := #MEC_GUA,
           ERROR_TIEMPO :=
         );

         CALL  #Maniobra_MC
         ( RESET        := TRUE,
           FIN_MANIOBRA := ,
           TIEMPO_LIM   := ,
           ACTUADOR     := ,
           B_FIN        := #MEC_MC,
           ERROR_TIEMPO :=
         );

         CALL  #Maniobra_ML
         ( RESET        := TRUE,
           FIN_MANIOBRA := ,
           TIEMPO_LIM   := ,
           ACTUADOR     := ,
           B_FIN        := #MEC_ML,
           ERROR_TIEMPO :=
         );



   _ERRLO:NOP   0;
END_REGION

REGION Network 4 (STL): DESCONEXIÓN POR ERROR REFRIGERANTE EN CNC
   // Desconexión por error en el tanque de refirgerante.
         A     #X38;

         R     #PARADA_ASINCRONA;
         S     #ERROR_REFRI;
         S     #PARADA_SINCRONA;
         R     #OFF_M;
         R     #ON_M;
         R     #AUTO_DIAG_CNC;

         JCN   _ERRRF;

         CALL  #Maniobra_Espada
         ( RESET        := TRUE,
           FIN_MANIOBRA := ,
           TIEMPO_LIM   := ,
           ACTUADOR     := #MEC_ESP,
           B_FIN        := ,
           ERROR_TIEMPO :=
         );

         CALL  #Maniobra_cuchillo
         ( RESET        := TRUE,
           FIN_MANIOBRA := ,
           TIEMPO_LIM   := ,
           ACTUADOR     := #MEC_CUC,
           B_FIN        := ,
           ERROR_TIEMPO :=
         );

         CALL  #Maniobra_katana
         ( RESET        := TRUE,
           FIN_MANIOBRA := ,
           TIEMPO_LIM   := ,
           ACTUADOR     := #MEC_KAT,
           B_FIN        := ,
           ERROR_TIEMPO :=
         );

         CALL  #Maniobra_florete
         ( RESET        := TRUE,
           FIN_MANIOBRA := ,
           TIEMPO_LIM   := ,
           ACTUADOR     := #MEC_FLO,
           B_FIN        := ,
           ERROR_TIEMPO :=
         );

         CALL  #Maniobra_sable
         ( RESET        := TRUE,
           FIN_MANIOBRA := ,
           TIEMPO_LIM   := ,
           ACTUADOR     := ,
           B_FIN        := #MEC_SAB,
           ERROR_TIEMPO :=
         );

         CALL  #Maniobra_hacha
         ( RESET        := TRUE,
           FIN_MANIOBRA := ,
           TIEMPO_LIM   := ,
           ACTUADOR     := ,
           B_FIN        := #MEC_HAC,
           ERROR_TIEMPO :=
         );

         CALL  #Maniobra_guada
         ( RESET        := TRUE,
           FIN_MANIOBRA := ,
           TIEMPO_LIM   := ,
           ACTUADOR     := ,
           B_FIN        := #MEC_GUA,
           ERROR_TIEMPO :=
         );

         CALL  #Maniobra_MC
         ( RESET        := TRUE,
           FIN_MANIOBRA := ,
           TIEMPO_LIM   := ,
           ACTUADOR     := ,
           B_FIN        := #MEC_MC,
           ERROR_TIEMPO :=
         );

         CALL  #Maniobra_ML
         ( RESET        := TRUE,
           FIN_MANIOBRA := ,
           TIEMPO_LIM   := ,
           ACTUADOR     := ,
           B_FIN        := #MEC_ML,
           ERROR_TIEMPO :=
         );



   _ERRRF:NOP   0;
END_REGION

REGION Network 5 (STL): DESCONEXIÓN POR ERROR TIEMPO EN CNC
   // Desconexión por error de tiempo durante el mecanizado.
         A     #X37;

         R     #PARADA_ASINCRONA;
         S     #ERROR_TIEMPO;
         S     #PARADA_SINCRONA;
         R     #OFF_M;
         R     #ON_M;
         R     #AUTO_DIAG_CNC;

         JCN   _ERRTMP;

         CALL  #Maniobra_Espada
         ( RESET        := TRUE,
           FIN_MANIOBRA := ,
           TIEMPO_LIM   := ,
           ACTUADOR     := #MEC_ESP,
           B_FIN        := ,
           ERROR_TIEMPO :=
         );

         CALL  #Maniobra_cuchillo
         ( RESET        := TRUE,
           FIN_MANIOBRA := ,
           TIEMPO_LIM   := ,
           ACTUADOR     := #MEC_CUC,
           B_FIN        := ,
           ERROR_TIEMPO :=
         );

         CALL  #Maniobra_katana
         ( RESET        := TRUE,
           FIN_MANIOBRA := ,
           TIEMPO_LIM   := ,
           ACTUADOR     := #MEC_KAT,
           B_FIN        := ,
           ERROR_TIEMPO :=
         );

         CALL  #Maniobra_florete
         ( RESET        := TRUE,
           FIN_MANIOBRA := ,
           TIEMPO_LIM   := ,
           ACTUADOR     := #MEC_FLO,
           B_FIN        := ,
           ERROR_TIEMPO :=
         );

         CALL  #Maniobra_sable
         ( RESET        := TRUE,
           FIN_MANIOBRA := ,
           TIEMPO_LIM   := ,
           ACTUADOR     := ,
           B_FIN        := #MEC_SAB,
           ERROR_TIEMPO :=
         );

         CALL  #Maniobra_hacha
         ( RESET        := TRUE,
           FIN_MANIOBRA := ,
           TIEMPO_LIM   := ,
           ACTUADOR     := ,
           B_FIN        := #MEC_HAC,
           ERROR_TIEMPO :=
         );

         CALL  #Maniobra_guada
         ( RESET        := TRUE,
           FIN_MANIOBRA := ,
           TIEMPO_LIM   := ,
           ACTUADOR     := ,
           B_FIN        := #MEC_GUA,
           ERROR_TIEMPO :=
         );

         CALL  #Maniobra_MC
         ( RESET        := TRUE,
           FIN_MANIOBRA := ,
           TIEMPO_LIM   := ,
           ACTUADOR     := ,
           B_FIN        := #MEC_MC,
           ERROR_TIEMPO :=
         );

         CALL  #Maniobra_ML
         ( RESET        := TRUE,
           FIN_MANIOBRA := ,
           TIEMPO_LIM   := ,
           ACTUADOR     := ,
           B_FIN        := #MEC_ML,
           ERROR_TIEMPO :=
         );



   _ERRTMP:NOP   0;
END_REGION

REGION Network 6 (STL): CONEXIÓN
   // Segmento de conexión de la CNC.
         A     #PETICION_CONEXION;
         FP    #B_TRABAJO;

         S     #X21;
         R     #X22;
         R     #X23;
         R     #X24;
         R     #X25;
         R     #X26;
         R     #X27;
         R     #X28;
         R     #X29;
         R     #X30;
         R     #X31;
         R     #X_APAGADO;
         R     #X35;
         R     #X36;
         R     #X37;
         R     #X38;

         S     #ON_M;
         R     #PARADA_ASINCRONA;
         R     #PARADA_SINCRONA;
         R     #ERROR_GLOBAL;
         R     #ERROR_LOCAL;
         R     #ERROR_TIEMPO;
         R     #ERROR_REFRI;
         R     #AUTO_DIAG_CNC;
         R     #OFF_M;


         JCN   _CONEXION;

         CALL  #Maniobra_Espada
         ( RESET        := TRUE,
           FIN_MANIOBRA := ,
           TIEMPO_LIM   := ,
           ACTUADOR     := #MEC_ESP,
           B_FIN        := ,
           ERROR_TIEMPO :=
         );

         CALL  #Maniobra_cuchillo
         ( RESET        := TRUE,
           FIN_MANIOBRA := ,
           TIEMPO_LIM   := ,
           ACTUADOR     := #MEC_CUC,
           B_FIN        := ,
           ERROR_TIEMPO :=
         );

         CALL  #Maniobra_katana
         ( RESET        := TRUE,
           FIN_MANIOBRA := ,
           TIEMPO_LIM   := ,
           ACTUADOR     := #MEC_KAT,
           B_FIN        := ,
           ERROR_TIEMPO :=
         );

         CALL  #Maniobra_florete
         ( RESET        := TRUE,
           FIN_MANIOBRA := ,
           TIEMPO_LIM   := ,
           ACTUADOR     := #MEC_FLO,
           B_FIN        := ,
           ERROR_TIEMPO :=
         );

         CALL  #Maniobra_sable
         ( RESET        := TRUE,
           FIN_MANIOBRA := ,
           TIEMPO_LIM   := ,
           ACTUADOR     := ,
           B_FIN        := #MEC_SAB,
           ERROR_TIEMPO :=
         );

         CALL  #Maniobra_hacha
         ( RESET        := TRUE,
           FIN_MANIOBRA := ,
           TIEMPO_LIM   := ,
           ACTUADOR     := ,
           B_FIN        := #MEC_HAC,
           ERROR_TIEMPO :=
         );

         CALL  #Maniobra_guada
         ( RESET        := TRUE,
           FIN_MANIOBRA := ,
           TIEMPO_LIM   := ,
           ACTUADOR     := ,
           B_FIN        := #MEC_GUA,
           ERROR_TIEMPO :=
         );

         CALL  #Maniobra_MC
         ( RESET        := TRUE,
           FIN_MANIOBRA := ,
           TIEMPO_LIM   := ,
           ACTUADOR     := ,
           B_FIN        := #MEC_MC,
           ERROR_TIEMPO :=
         );

         CALL  #Maniobra_ML
         ( RESET        := TRUE,
           FIN_MANIOBRA := ,
           TIEMPO_LIM   := ,
           ACTUADOR     := ,
           B_FIN        := #MEC_ML,
           ERROR_TIEMPO :=
         );


   _CONEXION:NOP   0;
END_REGION

REGION Network 7 (STL): CONGELACIÓN
         A     #MANT;

         =     #CONG_M;
         R     #AUTO_DIAG_CNC;
         R     #STANDBY_CNC;

         JCN   _CONGELACION;

         CALL  #Maniobra_Espada
         ( RESET        := TRUE,
           FIN_MANIOBRA := ,
           TIEMPO_LIM   := ,
           ACTUADOR     := #MEC_ESP,
           B_FIN        := ,
           ERROR_TIEMPO :=
         );

         CALL  #Maniobra_cuchillo
         ( RESET        := TRUE,
           FIN_MANIOBRA := ,
           TIEMPO_LIM   := ,
           ACTUADOR     := #MEC_CUC,
           B_FIN        := ,
           ERROR_TIEMPO :=
         );

         CALL  #Maniobra_katana
         ( RESET        := TRUE,
           FIN_MANIOBRA := ,
           TIEMPO_LIM   := ,
           ACTUADOR     := #MEC_KAT,
           B_FIN        := ,
           ERROR_TIEMPO :=
         );

         CALL  #Maniobra_florete
         ( RESET        := TRUE,
           FIN_MANIOBRA := ,
           TIEMPO_LIM   := ,
           ACTUADOR     := #MEC_FLO,
           B_FIN        := ,
           ERROR_TIEMPO :=
         );

         CALL  #Maniobra_sable
         ( RESET        := TRUE,
           FIN_MANIOBRA := ,
           TIEMPO_LIM   := ,
           ACTUADOR     := ,
           B_FIN        := #MEC_SAB,
           ERROR_TIEMPO :=
         );

         CALL  #Maniobra_hacha
         ( RESET        := TRUE,
           FIN_MANIOBRA := ,
           TIEMPO_LIM   := ,
           ACTUADOR     := ,
           B_FIN        := #MEC_HAC,
           ERROR_TIEMPO :=
         );

         CALL  #Maniobra_guada
         ( RESET        := TRUE,
           FIN_MANIOBRA := ,
           TIEMPO_LIM   := ,
           ACTUADOR     := ,
           B_FIN        := #MEC_GUA,
           ERROR_TIEMPO :=
         );

         CALL  #Maniobra_MC
         ( RESET        := TRUE,
           FIN_MANIOBRA := ,
           TIEMPO_LIM   := ,
           ACTUADOR     := ,
           B_FIN        := #MEC_MC,
           ERROR_TIEMPO :=
         );

         CALL  #Maniobra_ML
         ( RESET        := TRUE,
           FIN_MANIOBRA := ,
           TIEMPO_LIM   := ,
           ACTUADOR     := ,
           B_FIN        := #MEC_ML,
           ERROR_TIEMPO :=
         );


   _CONGELACION:NOP   0;

         A     #MANT;
         BEC;
END_REGION

REGION Network 8 (STL): ERROR ANALÓGICO REFRI
   // Medición del nivel del tanque de refrigerante.
         CALL  "Tratamiento_refrigerante"
         ( L_RAW     := #LIQUIDO_RAW,
           L_crit    := #L_crit,
           L_MIN     := #L_MIN,
           L_MAX     := #L_MAX,
           ERROR_LIM := #FLAG_REFRI,
           L_REAL    := #L_REAL,
           ERROR     := #ERROR_MEDICION
         );
END_REGION

REGION Network 9: REARME GLOBAL
   // Rearme tras emergencia global.
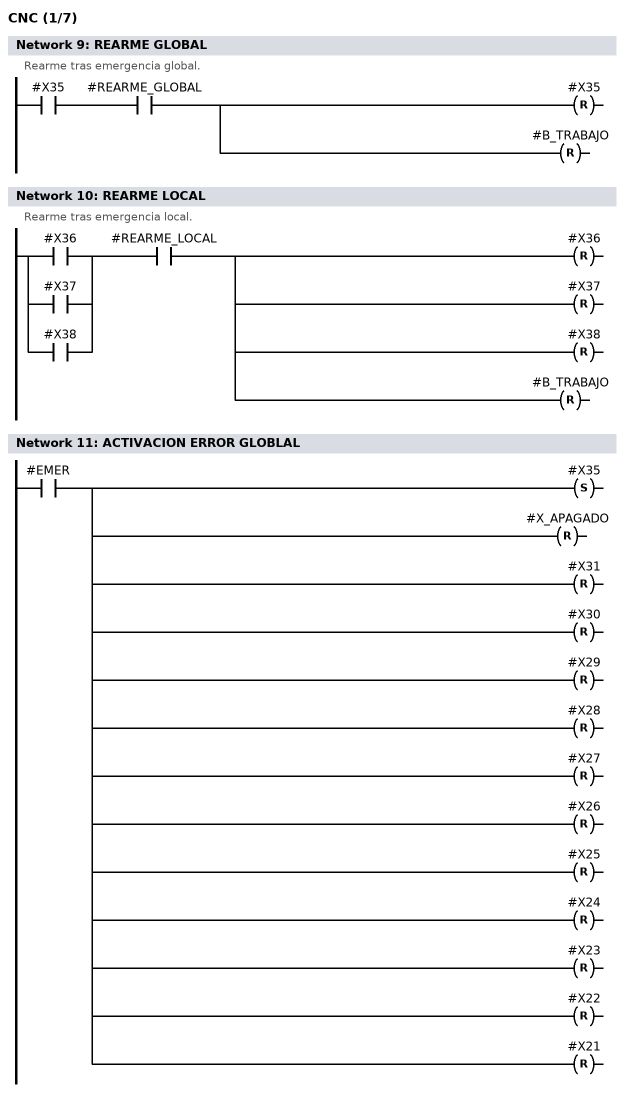
   RUNG wire#powerrail
      Contact( #X35 )
      Contact( #REARME_GLOBAL )
      wire#w1
      R_Coil( #X35 )
   END_RUNG
   RUNG wire#w1
      R_Coil( #B_TRABAJO )
   END_RUNG
   // the same network as SCL:
   #_w1 := #X35 AND #REARME_GLOBAL;
   IF #_w1 THEN
       #X35 := FALSE;
       #B_TRABAJO := FALSE;
   END_IF;
END_REGION

REGION Network 10: REARME LOCAL
   // Rearme tras emergencia local.
   RUNG wire#powerrail
      Contact( #X36 )
      wire#w1
      Contact( #REARME_LOCAL )
      wire#w2
      R_Coil( #X36 )
   END_RUNG
   RUNG wire#powerrail
      Contact( #X37 )
   END_RUNG wire#w1
   RUNG wire#powerrail
      Contact( #X38 )
   END_RUNG wire#w1
   RUNG wire#w2
      R_Coil( #X37 )
   END_RUNG
   RUNG wire#w2
      R_Coil( #X38 )
   END_RUNG
   RUNG wire#w2
      R_Coil( #B_TRABAJO )
   END_RUNG
   // the same network as SCL:
   #_w1 := (#X36 OR #X37 OR #X38) AND #REARME_LOCAL;
   IF #_w1 THEN
       #X36 := FALSE;
       #X37 := FALSE;
       #X38 := FALSE;
       #B_TRABAJO := FALSE;
   END_IF;
END_REGION

REGION Network 11: ACTIVACION ERROR GLOBLAL
   RUNG wire#powerrail
      Contact( #EMER )
      wire#w1
      S_Coil( #X35 )
   END_RUNG
   RUNG wire#w1
      R_Coil( #X_APAGADO )
   END_RUNG
   RUNG wire#w1
      R_Coil( #X31 )
   END_RUNG
   RUNG wire#w1
      R_Coil( #X30 )
   END_RUNG
   RUNG wire#w1
      R_Coil( #X29 )
   END_RUNG
   RUNG wire#w1
      R_Coil( #X28 )
   END_RUNG
   RUNG wire#w1
      R_Coil( #X27 )
   END_RUNG
   RUNG wire#w1
      R_Coil( #X26 )
   END_RUNG
   RUNG wire#w1
      R_Coil( #X25 )
   END_RUNG
   RUNG wire#w1
      R_Coil( #X24 )
   END_RUNG
   RUNG wire#w1
      R_Coil( #X23 )
   END_RUNG
   RUNG wire#w1
      R_Coil( #X22 )
   END_RUNG
   RUNG wire#w1
      R_Coil( #X21 )
   END_RUNG
   // the same network as SCL:
   IF #EMER THEN
       #X35 := TRUE;
       #X_APAGADO := FALSE;
       #X31 := FALSE;
       #X30 := FALSE;
       #X29 := FALSE;
       #X28 := FALSE;
       #X27 := FALSE;
       #X26 := FALSE;
       #X25 := FALSE;
       #X24 := FALSE;
       #X23 := FALSE;
       #X22 := FALSE;
       #X21 := FALSE;
   END_IF;
END_REGION

REGION Network 12: ERROR LOCAL
   // Activación del error en el autodiagnóstico o en la medición.
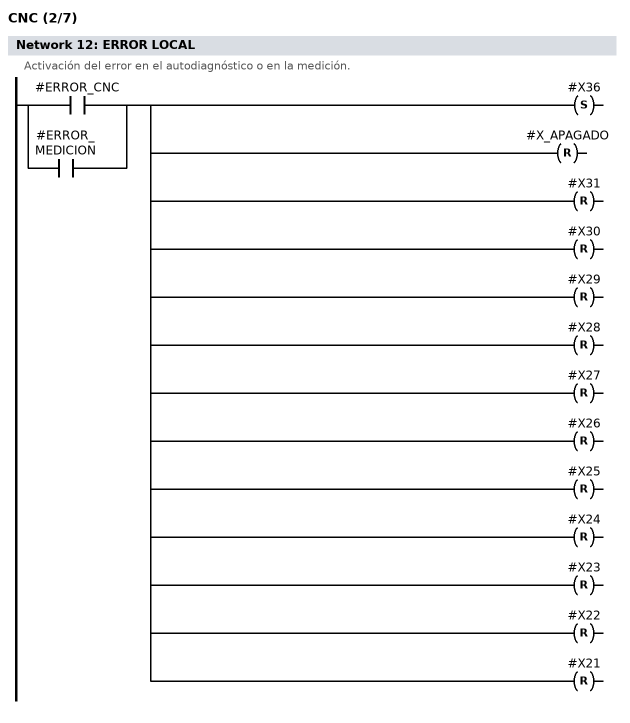
   RUNG wire#powerrail
      Contact( #ERROR_CNC )
      wire#w1
      S_Coil( #X36 )
   END_RUNG
   RUNG wire#powerrail
      Contact( #ERROR_MEDICION )
   END_RUNG wire#w1
   RUNG wire#w1
      R_Coil( #X_APAGADO )
   END_RUNG
   RUNG wire#w1
      R_Coil( #X31 )
   END_RUNG
   RUNG wire#w1
      R_Coil( #X30 )
   END_RUNG
   RUNG wire#w1
      R_Coil( #X29 )
   END_RUNG
   RUNG wire#w1
      R_Coil( #X28 )
   END_RUNG
   RUNG wire#w1
      R_Coil( #X27 )
   END_RUNG
   RUNG wire#w1
      R_Coil( #X26 )
   END_RUNG
   RUNG wire#w1
      R_Coil( #X25 )
   END_RUNG
   RUNG wire#w1
      R_Coil( #X24 )
   END_RUNG
   RUNG wire#w1
      R_Coil( #X23 )
   END_RUNG
   RUNG wire#w1
      R_Coil( #X22 )
   END_RUNG
   RUNG wire#w1
      R_Coil( #X21 )
   END_RUNG
   // the same network as SCL:
   IF #ERROR_CNC OR #ERROR_MEDICION THEN
       #X36 := TRUE;
       #X_APAGADO := FALSE;
       #X31 := FALSE;
       #X30 := FALSE;
       #X29 := FALSE;
       #X28 := FALSE;
       #X27 := FALSE;
       #X26 := FALSE;
       #X25 := FALSE;
       #X24 := FALSE;
       #X23 := FALSE;
       #X22 := FALSE;
       #X21 := FALSE;
   END_IF;
END_REGION

REGION Network 13: ERROR REFRI
   // Activación del error en el refrigerante.
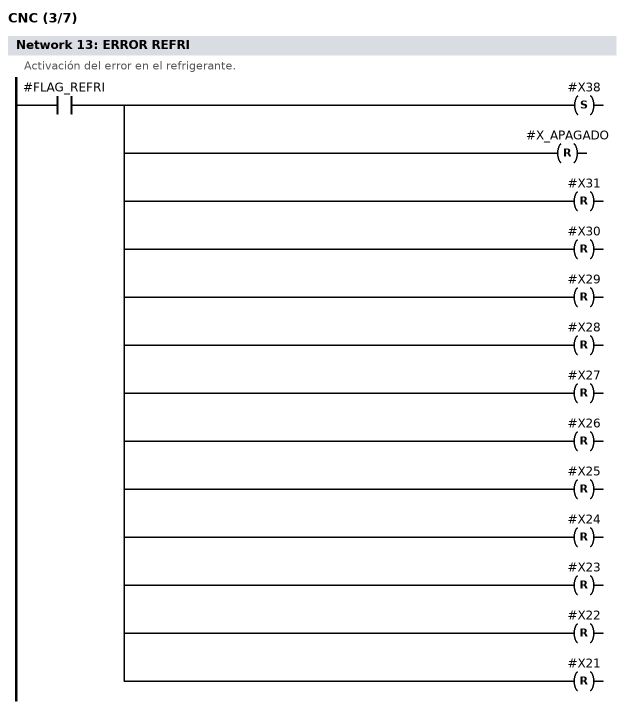
   RUNG wire#powerrail
      Contact( #FLAG_REFRI )
      wire#w1
      S_Coil( #X38 )
   END_RUNG
   RUNG wire#w1
      R_Coil( #X_APAGADO )
   END_RUNG
   RUNG wire#w1
      R_Coil( #X31 )
   END_RUNG
   RUNG wire#w1
      R_Coil( #X30 )
   END_RUNG
   RUNG wire#w1
      R_Coil( #X29 )
   END_RUNG
   RUNG wire#w1
      R_Coil( #X28 )
   END_RUNG
   RUNG wire#w1
      R_Coil( #X27 )
   END_RUNG
   RUNG wire#w1
      R_Coil( #X26 )
   END_RUNG
   RUNG wire#w1
      R_Coil( #X25 )
   END_RUNG
   RUNG wire#w1
      R_Coil( #X24 )
   END_RUNG
   RUNG wire#w1
      R_Coil( #X23 )
   END_RUNG
   RUNG wire#w1
      R_Coil( #X22 )
   END_RUNG
   RUNG wire#w1
      R_Coil( #X21 )
   END_RUNG
   // the same network as SCL:
   IF #FLAG_REFRI THEN
       #X38 := TRUE;
       #X_APAGADO := FALSE;
       #X31 := FALSE;
       #X30 := FALSE;
       #X29 := FALSE;
       #X28 := FALSE;
       #X27 := FALSE;
       #X26 := FALSE;
       #X25 := FALSE;
       #X24 := FALSE;
       #X23 := FALSE;
       #X22 := FALSE;
       #X21 := FALSE;
   END_IF;
END_REGION

REGION Network 14: ERROR TIEMPOS
   // Activación del error por exceso de tiempo.
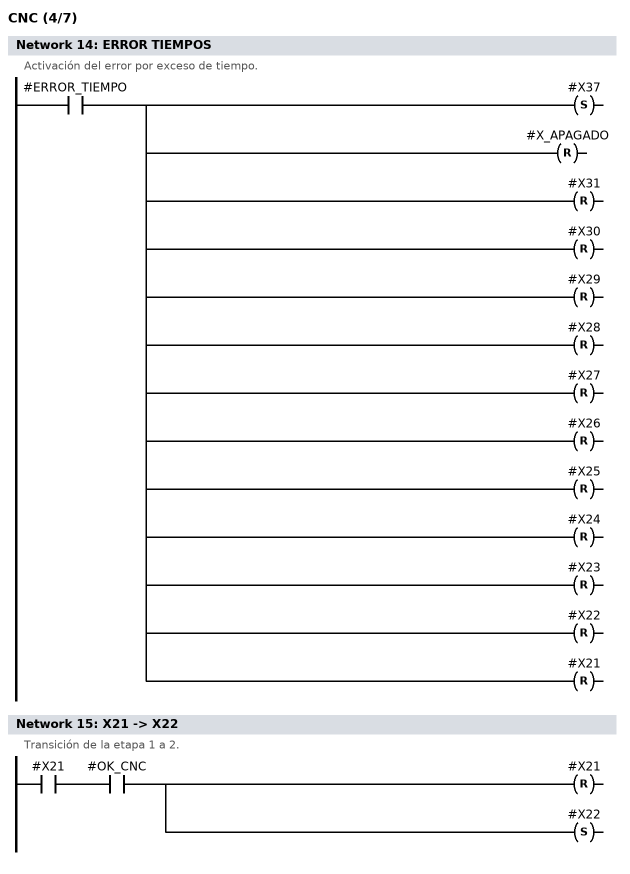
   RUNG wire#powerrail
      Contact( #ERROR_TIEMPO )
      wire#w1
      S_Coil( #X37 )
   END_RUNG
   RUNG wire#w1
      R_Coil( #X_APAGADO )
   END_RUNG
   RUNG wire#w1
      R_Coil( #X31 )
   END_RUNG
   RUNG wire#w1
      R_Coil( #X30 )
   END_RUNG
   RUNG wire#w1
      R_Coil( #X29 )
   END_RUNG
   RUNG wire#w1
      R_Coil( #X28 )
   END_RUNG
   RUNG wire#w1
      R_Coil( #X27 )
   END_RUNG
   RUNG wire#w1
      R_Coil( #X26 )
   END_RUNG
   RUNG wire#w1
      R_Coil( #X25 )
   END_RUNG
   RUNG wire#w1
      R_Coil( #X24 )
   END_RUNG
   RUNG wire#w1
      R_Coil( #X23 )
   END_RUNG
   RUNG wire#w1
      R_Coil( #X22 )
   END_RUNG
   RUNG wire#w1
      R_Coil( #X21 )
   END_RUNG
   // the same network as SCL:
   IF #ERROR_TIEMPO THEN
       #X37 := TRUE;
       #X_APAGADO := FALSE;
       #X31 := FALSE;
       #X30 := FALSE;
       #X29 := FALSE;
       #X28 := FALSE;
       #X27 := FALSE;
       #X26 := FALSE;
       #X25 := FALSE;
       #X24 := FALSE;
       #X23 := FALSE;
       #X22 := FALSE;
       #X21 := FALSE;
   END_IF;
END_REGION

REGION Network 15: X21 -> X22
   // Transición de la etapa 1 a 2.
   RUNG wire#powerrail
      Contact( #X21 )
      Contact( #OK_CNC )
      wire#w1
      R_Coil( #X21 )
   END_RUNG
   RUNG wire#w1
      S_Coil( #X22 )
   END_RUNG
   // the same network as SCL:
   #_w1 := #X21 AND #OK_CNC;
   IF #_w1 THEN
       #X21 := FALSE;
       #X22 := TRUE;
   END_IF;
END_REGION

REGION Network 16: SELECCION PIEZA
   // Divergencia OR para selección del tipo de mecanizado.
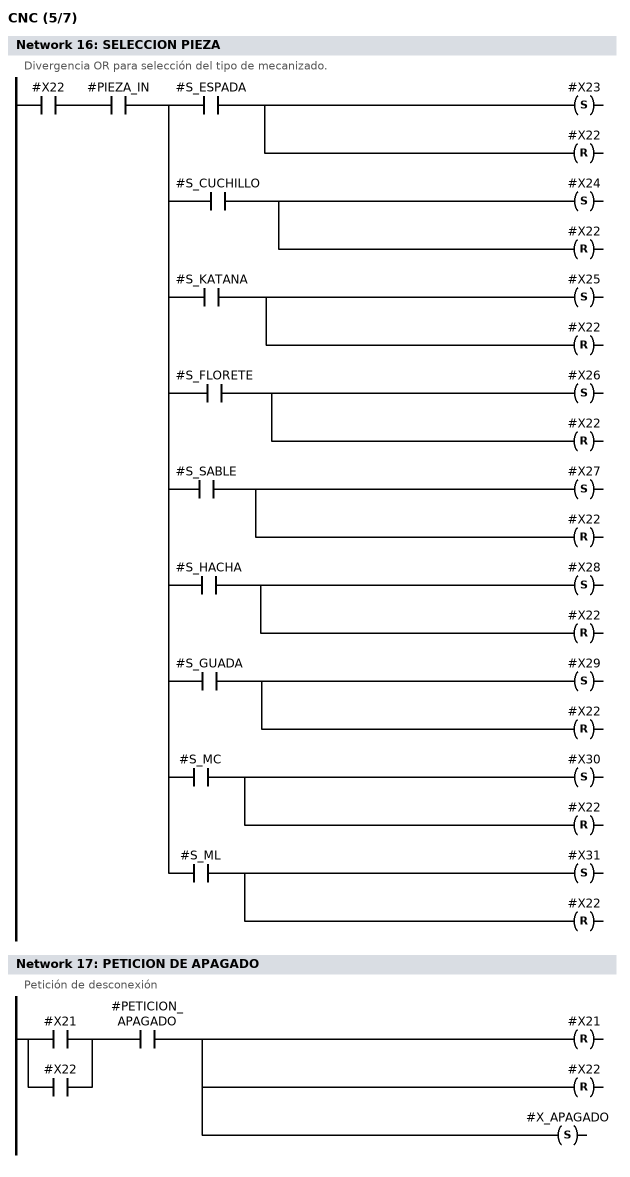
   RUNG wire#powerrail
      Contact( #X22 )
      Contact( #PIEZA_IN )
      wire#w1
      Contact( #S_ESPADA )
      wire#w2
      S_Coil( #X23 )
   END_RUNG
   RUNG wire#w2
      R_Coil( #X22 )
   END_RUNG
   RUNG wire#w1
      Contact( #S_CUCHILLO )
      wire#w3
      S_Coil( #X24 )
   END_RUNG
   RUNG wire#w3
      R_Coil( #X22 )
   END_RUNG
   RUNG wire#w1
      Contact( #S_KATANA )
      wire#w4
      S_Coil( #X25 )
   END_RUNG
   RUNG wire#w4
      R_Coil( #X22 )
   END_RUNG
   RUNG wire#w1
      Contact( #S_FLORETE )
      wire#w5
      S_Coil( #X26 )
   END_RUNG
   RUNG wire#w5
      R_Coil( #X22 )
   END_RUNG
   RUNG wire#w1
      Contact( #S_SABLE )
      wire#w6
      S_Coil( #X27 )
   END_RUNG
   RUNG wire#w6
      R_Coil( #X22 )
   END_RUNG
   RUNG wire#w1
      Contact( #S_HACHA )
      wire#w7
      S_Coil( #X28 )
   END_RUNG
   RUNG wire#w7
      R_Coil( #X22 )
   END_RUNG
   RUNG wire#w1
      Contact( #S_GUADA )
      wire#w8
      S_Coil( #X29 )
   END_RUNG
   RUNG wire#w8
      R_Coil( #X22 )
   END_RUNG
   RUNG wire#w1
      Contact( #S_MC )
      wire#w9
      S_Coil( #X30 )
   END_RUNG
   RUNG wire#w9
      R_Coil( #X22 )
   END_RUNG
   RUNG wire#w1
      Contact( #S_ML )
      wire#w10
      S_Coil( #X31 )
   END_RUNG
   RUNG wire#w10
      R_Coil( #X22 )
   END_RUNG
   // the same network as SCL:
   #_w1 := #X22 AND #PIEZA_IN;
   IF #_w1 AND #S_ESPADA THEN
       #X23 := TRUE;
       #X22 := FALSE;
   END_IF;
   IF #_w1 AND #S_CUCHILLO THEN
       #X24 := TRUE;
       #X22 := FALSE;
   END_IF;
   IF #_w1 AND #S_KATANA THEN
       #X25 := TRUE;
       #X22 := FALSE;
   END_IF;
   IF #_w1 AND #S_FLORETE THEN
       #X26 := TRUE;
       #X22 := FALSE;
   END_IF;
   IF #_w1 AND #S_SABLE THEN
       #X27 := TRUE;
       #X22 := FALSE;
   END_IF;
   IF #_w1 AND #S_HACHA THEN
       #X28 := TRUE;
       #X22 := FALSE;
   END_IF;
   IF #_w1 AND #S_GUADA THEN
       #X29 := TRUE;
       #X22 := FALSE;
   END_IF;
   IF #_w1 AND #S_MC THEN
       #X30 := TRUE;
       #X22 := FALSE;
   END_IF;
   IF #_w1 AND #S_ML THEN
       #X31 := TRUE;
       #X22 := FALSE;
   END_IF;
END_REGION

REGION Network 17: PETICION DE APAGADO
   // Petición de desconexión
   RUNG wire#powerrail
      Contact( #X21 )
      wire#w1
      Contact( #PETICION_APAGADO )
      wire#w2
      R_Coil( #X21 )
   END_RUNG
   RUNG wire#powerrail
      Contact( #X22 )
   END_RUNG wire#w1
   RUNG wire#w2
      R_Coil( #X22 )
   END_RUNG
   RUNG wire#w2
      S_Coil( #X_APAGADO )
   END_RUNG
   // the same network as SCL:
   #_w1 := (#X21 OR #X22) AND #PETICION_APAGADO;
   IF #_w1 THEN
       #X21 := FALSE;
       #X22 := FALSE;
       #X_APAGADO := TRUE;
   END_IF;
END_REGION

REGION Network 18: MECESP
   // Tratamiento de la etapa 23.
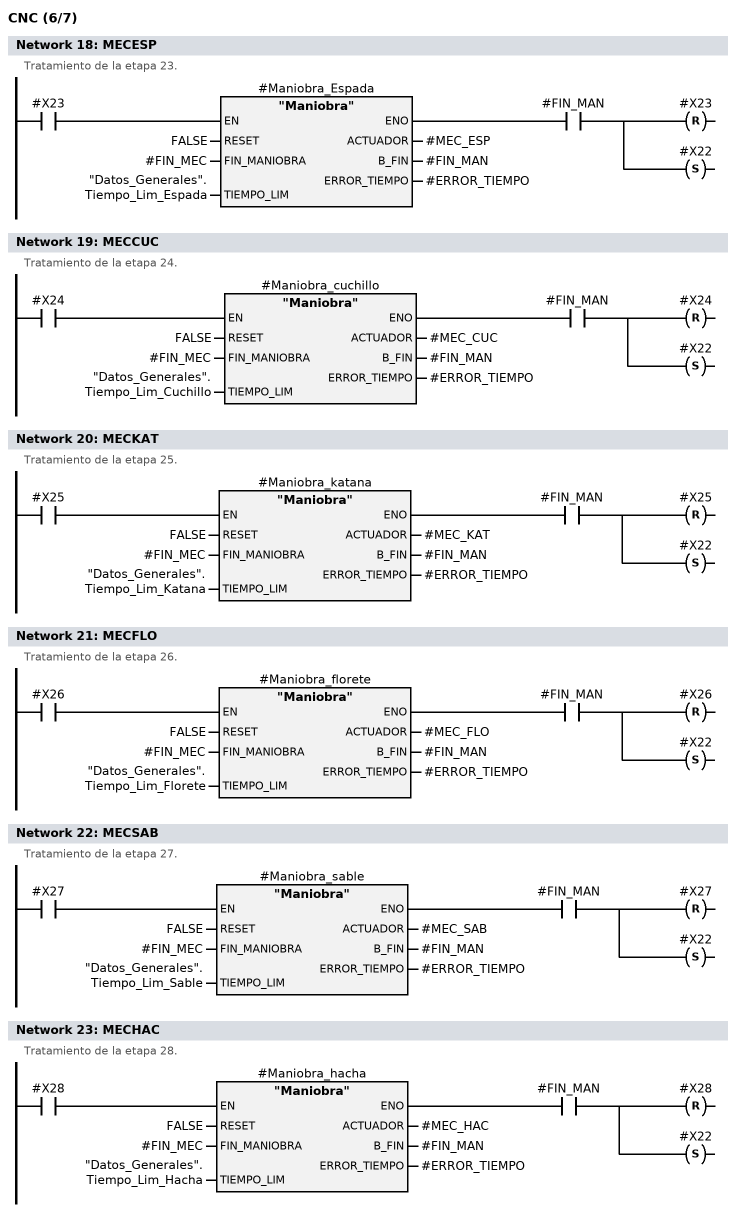
   RUNG wire#powerrail
      Contact( #X23 )
      #Maniobra_Espada(RESET := FALSE, FIN_MANIOBRA := #FIN_MEC, TIEMPO_LIM := "Datos_Generales".Tiempo_Lim_Espada, ACTUADOR => #MEC_ESP, B_FIN => #FIN_MAN, ERROR_TIEMPO => #ERROR_TIEMPO)
      Contact( #FIN_MAN )
      wire#w1
      R_Coil( #X23 )
   END_RUNG
   RUNG wire#w1
      S_Coil( #X22 )
   END_RUNG
   // the same network as SCL:
   #Maniobra_Espada(EN := #X23,   // "Maniobra"
                    RESET := FALSE,
                    FIN_MANIOBRA := #FIN_MEC,
                    TIEMPO_LIM := "Datos_Generales".Tiempo_Lim_Espada,
                    ACTUADOR => #MEC_ESP,
                    B_FIN => #FIN_MAN,
                    ERROR_TIEMPO => #ERROR_TIEMPO,
                    ENO => #_w1);
   IF #_w1 AND #FIN_MAN THEN
       #X23 := FALSE;
       #X22 := TRUE;
   END_IF;
END_REGION

REGION Network 19: MECCUC
   // Tratamiento de la etapa 24.
   RUNG wire#powerrail
      Contact( #X24 )
      #Maniobra_cuchillo(RESET := FALSE, FIN_MANIOBRA := #FIN_MEC, TIEMPO_LIM := "Datos_Generales".Tiempo_Lim_Cuchillo, ACTUADOR => #MEC_CUC, B_FIN => #FIN_MAN, ERROR_TIEMPO => #ERROR_TIEMPO)
      Contact( #FIN_MAN )
      wire#w1
      R_Coil( #X24 )
   END_RUNG
   RUNG wire#w1
      S_Coil( #X22 )
   END_RUNG
   // the same network as SCL:
   #Maniobra_cuchillo(EN := #X24,   // "Maniobra"
                      RESET := FALSE,
                      FIN_MANIOBRA := #FIN_MEC,
                      TIEMPO_LIM := "Datos_Generales".Tiempo_Lim_Cuchillo,
                      ACTUADOR => #MEC_CUC,
                      B_FIN => #FIN_MAN,
                      ERROR_TIEMPO => #ERROR_TIEMPO,
                      ENO => #_w1);
   IF #_w1 AND #FIN_MAN THEN
       #X24 := FALSE;
       #X22 := TRUE;
   END_IF;
END_REGION

REGION Network 20: MECKAT
   // Tratamiento de la etapa 25.
   RUNG wire#powerrail
      Contact( #X25 )
      #Maniobra_katana(RESET := FALSE, FIN_MANIOBRA := #FIN_MEC, TIEMPO_LIM := "Datos_Generales".Tiempo_Lim_Katana, ACTUADOR => #MEC_KAT, B_FIN => #FIN_MAN, ERROR_TIEMPO => #ERROR_TIEMPO)
      Contact( #FIN_MAN )
      wire#w1
      R_Coil( #X25 )
   END_RUNG
   RUNG wire#w1
      S_Coil( #X22 )
   END_RUNG
   // the same network as SCL:
   #Maniobra_katana(EN := #X25,   // "Maniobra"
                    RESET := FALSE,
                    FIN_MANIOBRA := #FIN_MEC,
                    TIEMPO_LIM := "Datos_Generales".Tiempo_Lim_Katana,
                    ACTUADOR => #MEC_KAT,
                    B_FIN => #FIN_MAN,
                    ERROR_TIEMPO => #ERROR_TIEMPO,
                    ENO => #_w1);
   IF #_w1 AND #FIN_MAN THEN
       #X25 := FALSE;
       #X22 := TRUE;
   END_IF;
END_REGION

REGION Network 21: MECFLO
   // Tratamiento de la etapa 26.
   RUNG wire#powerrail
      Contact( #X26 )
      #Maniobra_florete(RESET := FALSE, FIN_MANIOBRA := #FIN_MEC, TIEMPO_LIM := "Datos_Generales".Tiempo_Lim_Florete, ACTUADOR => #MEC_FLO, B_FIN => #FIN_MAN, ERROR_TIEMPO => #ERROR_TIEMPO)
      Contact( #FIN_MAN )
      wire#w1
      R_Coil( #X26 )
   END_RUNG
   RUNG wire#w1
      S_Coil( #X22 )
   END_RUNG
   // the same network as SCL:
   #Maniobra_florete(EN := #X26,   // "Maniobra"
                     RESET := FALSE,
                     FIN_MANIOBRA := #FIN_MEC,
                     TIEMPO_LIM := "Datos_Generales".Tiempo_Lim_Florete,
                     ACTUADOR => #MEC_FLO,
                     B_FIN => #FIN_MAN,
                     ERROR_TIEMPO => #ERROR_TIEMPO,
                     ENO => #_w1);
   IF #_w1 AND #FIN_MAN THEN
       #X26 := FALSE;
       #X22 := TRUE;
   END_IF;
END_REGION

REGION Network 22: MECSAB
   // Tratamiento de la etapa 27.
   RUNG wire#powerrail
      Contact( #X27 )
      #Maniobra_sable(RESET := FALSE, FIN_MANIOBRA := #FIN_MEC, TIEMPO_LIM := "Datos_Generales".Tiempo_Lim_Sable, ACTUADOR => #MEC_SAB, B_FIN => #FIN_MAN, ERROR_TIEMPO => #ERROR_TIEMPO)
      Contact( #FIN_MAN )
      wire#w1
      R_Coil( #X27 )
   END_RUNG
   RUNG wire#w1
      S_Coil( #X22 )
   END_RUNG
   // the same network as SCL:
   #Maniobra_sable(EN := #X27,   // "Maniobra"
                   RESET := FALSE,
                   FIN_MANIOBRA := #FIN_MEC,
                   TIEMPO_LIM := "Datos_Generales".Tiempo_Lim_Sable,
                   ACTUADOR => #MEC_SAB,
                   B_FIN => #FIN_MAN,
                   ERROR_TIEMPO => #ERROR_TIEMPO,
                   ENO => #_w1);
   IF #_w1 AND #FIN_MAN THEN
       #X27 := FALSE;
       #X22 := TRUE;
   END_IF;
END_REGION

REGION Network 23: MECHAC
   // Tratamiento de la etapa 28.
   RUNG wire#powerrail
      Contact( #X28 )
      #Maniobra_hacha(RESET := FALSE, FIN_MANIOBRA := #FIN_MEC, TIEMPO_LIM := "Datos_Generales".Tiempo_Lim_Hacha, ACTUADOR => #MEC_HAC, B_FIN => #FIN_MAN, ERROR_TIEMPO => #ERROR_TIEMPO)
      Contact( #FIN_MAN )
      wire#w1
      R_Coil( #X28 )
   END_RUNG
   RUNG wire#w1
      S_Coil( #X22 )
   END_RUNG
   // the same network as SCL:
   #Maniobra_hacha(EN := #X28,   // "Maniobra"
                   RESET := FALSE,
                   FIN_MANIOBRA := #FIN_MEC,
                   TIEMPO_LIM := "Datos_Generales".Tiempo_Lim_Hacha,
                   ACTUADOR => #MEC_HAC,
                   B_FIN => #FIN_MAN,
                   ERROR_TIEMPO => #ERROR_TIEMPO,
                   ENO => #_w1);
   IF #_w1 AND #FIN_MAN THEN
       #X28 := FALSE;
       #X22 := TRUE;
   END_IF;
END_REGION

REGION Network 24: MECGUA
   // Tratamiento de la etapa 29.
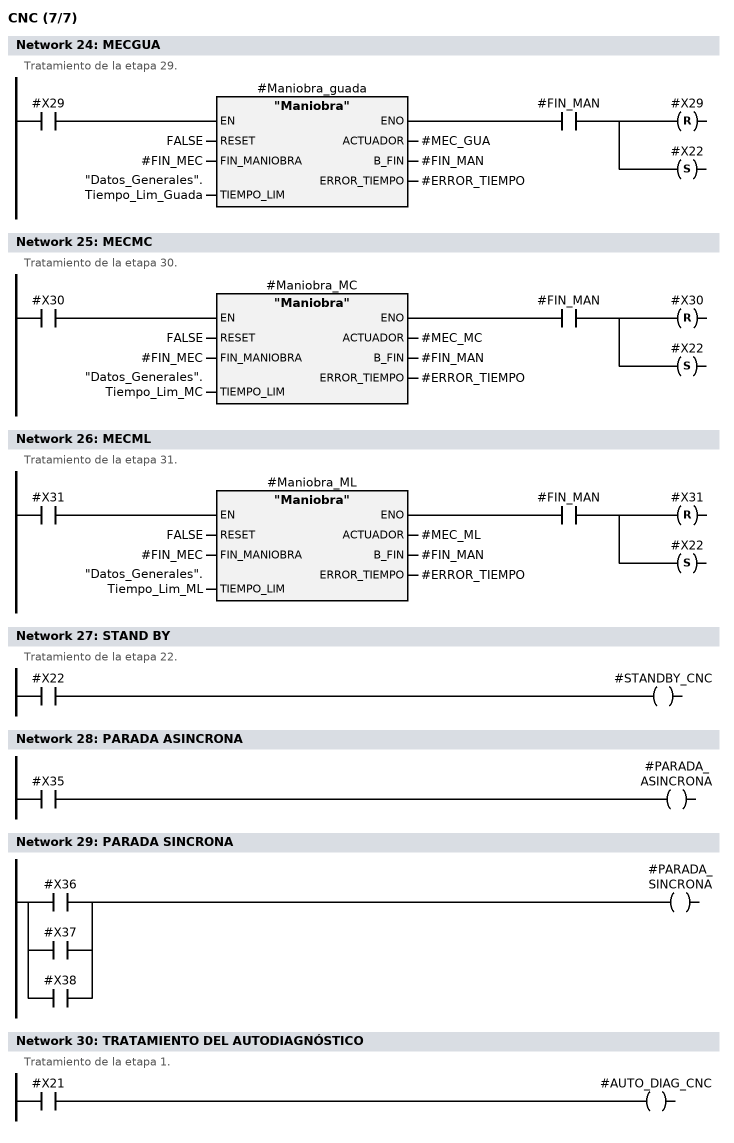
   RUNG wire#powerrail
      Contact( #X29 )
      #Maniobra_guada(RESET := FALSE, FIN_MANIOBRA := #FIN_MEC, TIEMPO_LIM := "Datos_Generales".Tiempo_Lim_Guada, ACTUADOR => #MEC_GUA, B_FIN => #FIN_MAN, ERROR_TIEMPO => #ERROR_TIEMPO)
      Contact( #FIN_MAN )
      wire#w1
      R_Coil( #X29 )
   END_RUNG
   RUNG wire#w1
      S_Coil( #X22 )
   END_RUNG
   // the same network as SCL:
   #Maniobra_guada(EN := #X29,   // "Maniobra"
                   RESET := FALSE,
                   FIN_MANIOBRA := #FIN_MEC,
                   TIEMPO_LIM := "Datos_Generales".Tiempo_Lim_Guada,
                   ACTUADOR => #MEC_GUA,
                   B_FIN => #FIN_MAN,
                   ERROR_TIEMPO => #ERROR_TIEMPO,
                   ENO => #_w1);
   IF #_w1 AND #FIN_MAN THEN
       #X29 := FALSE;
       #X22 := TRUE;
   END_IF;
END_REGION

REGION Network 25: MECMC
   // Tratamiento de la etapa 30.
   RUNG wire#powerrail
      Contact( #X30 )
      #Maniobra_MC(RESET := FALSE, FIN_MANIOBRA := #FIN_MEC, TIEMPO_LIM := "Datos_Generales".Tiempo_Lim_MC, ACTUADOR => #MEC_MC, B_FIN => #FIN_MAN, ERROR_TIEMPO => #ERROR_TIEMPO)
      Contact( #FIN_MAN )
      wire#w1
      R_Coil( #X30 )
   END_RUNG
   RUNG wire#w1
      S_Coil( #X22 )
   END_RUNG
   // the same network as SCL:
   #Maniobra_MC(EN := #X30,   // "Maniobra"
                RESET := FALSE,
                FIN_MANIOBRA := #FIN_MEC,
                TIEMPO_LIM := "Datos_Generales".Tiempo_Lim_MC,
                ACTUADOR => #MEC_MC,
                B_FIN => #FIN_MAN,
                ERROR_TIEMPO => #ERROR_TIEMPO,
                ENO => #_w1);
   IF #_w1 AND #FIN_MAN THEN
       #X30 := FALSE;
       #X22 := TRUE;
   END_IF;
END_REGION

REGION Network 26: MECML
   // Tratamiento de la etapa 31.
   RUNG wire#powerrail
      Contact( #X31 )
      #Maniobra_ML(RESET := FALSE, FIN_MANIOBRA := #FIN_MEC, TIEMPO_LIM := "Datos_Generales".Tiempo_Lim_ML, ACTUADOR => #MEC_ML, B_FIN => #FIN_MAN, ERROR_TIEMPO => #ERROR_TIEMPO)
      Contact( #FIN_MAN )
      wire#w1
      R_Coil( #X31 )
   END_RUNG
   RUNG wire#w1
      S_Coil( #X22 )
   END_RUNG
   // the same network as SCL:
   #Maniobra_ML(EN := #X31,   // "Maniobra"
                RESET := FALSE,
                FIN_MANIOBRA := #FIN_MEC,
                TIEMPO_LIM := "Datos_Generales".Tiempo_Lim_ML,
                ACTUADOR => #MEC_ML,
                B_FIN => #FIN_MAN,
                ERROR_TIEMPO => #ERROR_TIEMPO,
                ENO => #_w1);
   IF #_w1 AND #FIN_MAN THEN
       #X31 := FALSE;
       #X22 := TRUE;
   END_IF;
END_REGION

REGION Network 27: STAND BY
   // Tratamiento de la etapa 22.
   RUNG wire#powerrail
      Contact( #X22 )
      Coil( #STANDBY_CNC )
   END_RUNG
   // the same network as SCL:
   #STANDBY_CNC := #X22;
END_REGION

REGION Network 28: PARADA ASINCRONA
   RUNG wire#powerrail
      Contact( #X35 )
      Coil( #PARADA_ASINCRONA )
   END_RUNG
   // the same network as SCL:
   #PARADA_ASINCRONA := #X35;
END_REGION

REGION Network 29: PARADA SINCRONA
   RUNG wire#powerrail
      Contact( #X36 )
      wire#w1
      Coil( #PARADA_SINCRONA )
   END_RUNG
   RUNG wire#powerrail
      Contact( #X37 )
   END_RUNG wire#w1
   RUNG wire#powerrail
      Contact( #X38 )
   END_RUNG wire#w1
   // the same network as SCL:
   #PARADA_SINCRONA := #X36 OR #X37 OR #X38;
END_REGION

REGION Network 30: TRATAMIENTO DEL AUTODIAGNÓSTICO
   // Tratamiento de la etapa 1.
   RUNG wire#powerrail
      Contact( #X21 )
      Coil( #AUTO_DIAG_CNC )
   END_RUNG
   // the same network as SCL:
   #AUTO_DIAG_CNC := #X21;
END_REGION

REGION Network 31 (STL): APAGADO DE LA CNC
   // Apagado de la CNC.
         A     #X_APAGADO;
         S     #OFF_M;
         R     #ON_M;
         JCN   _PARADA;

         CALL  #Maniobra_Espada
         ( RESET        := TRUE,
           FIN_MANIOBRA := ,
           TIEMPO_LIM   := ,
           ACTUADOR     := #MEC_ESP,
           B_FIN        := ,
           ERROR_TIEMPO :=
         );

         CALL  #Maniobra_cuchillo
         ( RESET        := TRUE,
           FIN_MANIOBRA := ,
           TIEMPO_LIM   := ,
           ACTUADOR     := #MEC_CUC,
           B_FIN        := ,
           ERROR_TIEMPO :=
         );

         CALL  #Maniobra_katana
         ( RESET        := TRUE,
           FIN_MANIOBRA := ,
           TIEMPO_LIM   := ,
           ACTUADOR     := #MEC_KAT,
           B_FIN        := ,
           ERROR_TIEMPO :=
         );

         CALL  #Maniobra_florete
         ( RESET        := TRUE,
           FIN_MANIOBRA := ,
           TIEMPO_LIM   := ,
           ACTUADOR     := #MEC_FLO,
           B_FIN        := ,
           ERROR_TIEMPO :=
         );

         CALL  #Maniobra_sable
         ( RESET        := TRUE,
           FIN_MANIOBRA := ,
           TIEMPO_LIM   := ,
           ACTUADOR     := ,
           B_FIN        := #MEC_SAB,
           ERROR_TIEMPO :=
         );

         CALL  #Maniobra_hacha
         ( RESET        := TRUE,
           FIN_MANIOBRA := ,
           TIEMPO_LIM   := ,
           ACTUADOR     := ,
           B_FIN        := #MEC_HAC,
           ERROR_TIEMPO :=
         );

         CALL  #Maniobra_guada
         ( RESET        := TRUE,
           FIN_MANIOBRA := ,
           TIEMPO_LIM   := ,
           ACTUADOR     := ,
           B_FIN        := #MEC_GUA,
           ERROR_TIEMPO :=
         );

         CALL  #Maniobra_MC
         ( RESET        := TRUE,
           FIN_MANIOBRA := ,
           TIEMPO_LIM   := ,
           ACTUADOR     := ,
           B_FIN        := #MEC_MC,
           ERROR_TIEMPO :=
         );

         CALL  #Maniobra_ML
         ( RESET        := TRUE,
           FIN_MANIOBRA := ,
           TIEMPO_LIM   := ,
           ACTUADOR     := ,
           B_FIN        := #MEC_ML,
           ERROR_TIEMPO :=
         );

         CALL  #Maniobra_APAGADO
         ( RESET        := FALSE,
           FIN_MANIOBRA := #APAGADO_CONFIRMADO,
           TIEMPO_LIM   := #TIEMPO_LIM,
           ACTUADOR     := #APAGADO_CNC,
           B_FIN        := #FIN_PARADA,
           ERROR_TIEMPO := #ERROR_TIEMPO
         );

         A     #FIN_PARADA;
         S     #X_FIN;
         R     #X_APAGADO;

         A     #ERROR_TIEMPO;
         S     #X37;
         R     #X_APAGADO;


   _PARADA:NOP   0;
END_REGION
END_FUNCTION_BLOCK

FUNCTION_BLOCK "Celda_Mecanizado"   // FB5, STL
{ S7_Optimized_Access := 'TRUE' }
VERSION : 0.1
BEGIN
END_FUNCTION_BLOCK

FUNCTION "Tratamiento_velocidad" : Void   // FC1, STL
TITLE = Conectores de la señal analógica.
{ S7_Optimized_Access := 'TRUE' }
VERSION : 0.1
// En este bloque se comparará la velocidad del motor con la que debería tener.
   VAR_INPUT
      V_RAW : Int;   // Valor de la señal desde el sensor.
      V_med : Real;   // Velocidad permanente que se quiere comparar.
      V_MIN : Real;   // Mínimo de velocidad que se puede medir.
      V_MAX : Real;   // Máximo de velocidad que se puede medir.
      V_MAX_ADM : Real;   // Máxima velocidad admitida en régimen permanente.
      V_MIN_ADM : Real;   // Mínima velocidad permitida en régimen permanente.
   END_VAR
   VAR_OUTPUT
      V_baja : Bool;   // La velocidad es muy lenta.
      V_alta : Bool;   // La velocidad es muy rápida.
      V_parada : Bool;   // Está parado.
      V_OK_SUBIDA : Bool;   // Velocidad alcanzada acelerando.
      V_OK_BAJADA : Bool;   // Velocidad alcanzada frenando.
   END_VAR
   VAR_IN_OUT
      V_REAL : Real;   // Velocidad real del motor.
      ERROR : Bool;   // Error durante la medición.
   END_VAR
BEGIN

REGION Network 1: Tratamiento de la señal analógica.
   // Conversión dela señal medida por el sensor.
         CALL  "Tratamiento_analogico"
         ( raw_vel     := #V_RAW,
           V_min       := #V_MIN,
           V_max       := #V_MAX,
           V           := #V_REAL,
           aviso_error := #ERROR
         );
END_REGION

REGION Network 2: Error durante la medición.
   // Si hay un error en la medición se sale del bloque.
         A     #ERROR;
         BEC;
END_REGION

REGION Network 3: Comparación de velocidades.
   // Se compara si la velocidad es baja.
         L     #V_REAL;
         L     #V_MIN_ADM;
         <R;
         =     #V_baja;
END_REGION

REGION Network 4: Comparación de velocidades.
   // Se compara si la velocidad es alta.
         L     #V_REAL;
         L     #V_MAX_ADM;
         >R;
         =     #V_alta;
END_REGION

REGION Network 5: Comparación de velocidades.
   // Se compara si la velocidad es 0.
         L     #V_REAL;
         L     0.0;
         ==R;
         =     #V_parada;
END_REGION

REGION Network 6: Velocidad OK de subida.
   // Se ha acelerado al régimen aceptable.
         L     #V_REAL;
         L     #V_med;
         >R;
         =     #V_OK_SUBIDA;
END_REGION

REGION Network 7: Velocidad OK de bajada.
   // Se ha frenado al régimen aceptable.
         A     <0;
         =     #V_OK_BAJADA;
END_REGION
END_FUNCTION

FUNCTION "Tratamiento_analogico" : Void   // FC2, STL
TITLE = TRATAMIENTO ANALÓGICO
{ S7_Optimized_Access := 'TRUE' }
VERSION : 0.1
// Este bloque se encarga del tratamiento de la señal analógica.
   VAR_INPUT
      raw_vel : Int;   // Velocidad digitalizada del sensor.
      V_min : Real;   // Mínimo de velocidad que se puede medir.
      V_max : Real;   // Máximo de velocidad que se puede medir.
   END_VAR
   VAR_OUTPUT
      V : Real;   // Velocidad analógica convertida.
      aviso_error : Bool;   // Error durante tratamiento.
   END_VAR
   VAR_TEMP
      ret_val_1 : Word;   // Error.
   END_VAR
BEGIN

REGION Network 1: SEÑAL ANALÓGICA
   // Conversión de la señal de entrada a un valor real.
         CALL  SCALE
         ( IN      := #raw_vel,
           HI_LIM  := #V_max,
           LO_LIM  := #V_min,
           BIPOLAR := FALSE,
           RET_VAL := #ret_val_1,
           OUT     := #V
         );
END_REGION

REGION Network 2: GESTIÓN DEL ERROR
   // Si ret_val_1 es 0, la medida es correcta. Si no da error.
         L     #ret_val_1;
         L     0;
         <>I;
         =     #aviso_error;
END_REGION
END_FUNCTION

FUNCTION "Tratamiento_refrigerante" : Void   // FC3, STL
TITLE = Conectores de la señal analógica.
{ S7_Optimized_Access := 'TRUE' }
VERSION : 0.1
// En este bloque se comparará la velocidad del motor con la que debería tener.
   VAR_INPUT
      L_RAW : Int;   // Valor de la señal desde el sensor.
      L_crit : Real;   // Valor de refrigerante crítico.
      L_MIN : Real;   // Mínimo de refrigerante que se puede medir.
      L_MAX : Real;   // Máximo de refrigerante que se puede medir.
   END_VAR
   VAR_OUTPUT
      ERROR_LIM : Bool;   // Error por límite del refrigerante.
   END_VAR
   VAR_IN_OUT
      L_REAL : Real;   // Nivel de refrigerante real de la CNC.
      ERROR : Bool;   // Error durante la medición.
   END_VAR
BEGIN

REGION Network 1: Tratamiento de la señal analógica.
   // Conversión dela señal medida por el sensor.
         CALL  "Tratamiento_analogico"
         ( raw_vel     := #L_RAW,
           V_min       := #L_MIN,
           V_max       := #L_MAX,
           V           := #L_REAL,
           aviso_error := #ERROR
         );
END_REGION

REGION Network 2: Error durante la medición.
   // Si hay un error en la medición se sale del bloque.
         A     #ERROR;
         BEC;
END_REGION

REGION Network 3: Error por límite del refrigerante.
   // Si el nivel de refrigerante pasa por debajo de un mínimo salta el error.
         L     #L_REAL;
         L     #L_crit;
         <R;
         =     #ERROR_LIM;
END_REGION
END_FUNCTION

FUNCTION "RFID" : Void   // FC4, STL
TITLE = RFID
{ S7_Optimized_Access := 'TRUE' }
VERSION : 0.1
// Este bloque simula la lectura de una tarjeta RFID. 
// Se leerán 5 bits. El primero indica el tipo de productos, mientras que el segundo trata el proceso siguiente al que tiene que ir.
   VAR_INPUT
      TIPO : Int;   // Tipo de arma.
      PROCESO : Int;   // Proceso siguiente al que tiene que ir.
   END_VAR
   VAR_IN_OUT
      S_ESPADA : Bool;   // Se trata de una espada.
      S_CUCHILLO : Bool;   // Se trata de un cuchillo.
      S_KATANA : Bool;   // Se trata de una katana.
      S_FLORETE : Bool;   // Se trata de un florete.
      S_SABLE : Bool;   // Se trata de un sable.
      S_HACHA : Bool;   // Se trata de un hacha.
      S_GUADAÑA : Bool;   // Se trata de una guadaña.
      S_MANGO_CORTO : Bool;   // Se trata de un mango corto.
      S_MANGO_LARGO : Bool;   // Se trata de un mango largo.
      DO_NOTHING : Bool;   // No toca mecanizar la pieza.
      MECANIZAR : Bool;   // La pieza debe ser mecanizada.
      SALIR : Bool;   // La pieza está lista para salir de la celda.
   END_VAR
BEGIN

REGION Network 1: Comprobación de S_Espada
   // En este segmento se comprobará si los bits leídos corresponden con la espada larga.
         L     #TIPO;
         L     0;
         ==I;
         =     #S_ESPADA;
END_REGION

REGION Network 2: Comprobación de S_Cuchillo
   // En este segmento se comprobará si los bits leídos corresponden con el cuchillo.
         L     #TIPO;
         L     1;
         ==I;
         =     #S_CUCHILLO;
END_REGION

REGION Network 3: Comprobación de S_Katana
   // En este segmento se comprobará si los bits leídos corresponden con la katana.
         L     #TIPO;
         L     2;
         ==I;
         =     #S_KATANA;
END_REGION

REGION Network 4: Comprobación de S_Florete
   // En este segmento se comprobará si los bits leídos corresponden con el florete.
         L     #TIPO;
         L     3;
         ==I;
         =     #S_FLORETE;
END_REGION

REGION Network 5: Comprobación de S_Sable
   // En este segmento se comprobará si los bits leídos corresponden con el sable.
         L     #TIPO;
         L     4;
         ==I;
         =     #S_SABLE;
END_REGION

REGION Network 6: Comprobación de S_Hacha
   // En este segmento se comprobará si los bits leídos corresponden con el hacha.
         L     #TIPO;
         L     5;
         ==I;
         =     #S_HACHA;
END_REGION

REGION Network 7: Comprobación de S_Guadaña
   // En este segmento se comprobará si los bits leídos corresponden con la guadaña.
         L     #TIPO;
         L     6;
         ==I;
         =     #S_GUADAÑA;
END_REGION

REGION Network 8: Comprobación de S_MangoCorto
   // En este segmento se comprobará si los bits leídos corresponden con el mango corto.
         L     #TIPO;
         L     7;
         ==I;
         =     #S_MANGO_CORTO;
END_REGION

REGION Network 9: Comprobación de S_Mango_Largo
   // En este segmento se comprobará si los bits leídos corresponden con el mango largo.
         L     #TIPO;
         L     8;
         ==I;
         =     #S_MANGO_LARGO;
END_REGION

REGION Network 10: Comprobación de proceso
   // Este segmento se encarga de determinar si el producto necesita pasar por el mecanizado o no
         L     #PROCESO;
         L     2;
         ==I;
         =     #MECANIZAR;
END_REGION

REGION Network 11: Comprobación de proceso
   // Este segmento se encarga de determinar si el producto necesita pasar por el mecanizado o no
         L     #PROCESO;
         L     3;
         ==I;
         =     #SALIR;
END_REGION

REGION Network 12: Comprobación de proceso
   // Este segmento se encarga de determinar si el producto necesita pasar por el mecanizado o no
         L     #PROCESO;
         L     2;
         <I;
         =     #DO_NOTHING;
END_REGION
END_FUNCTION